LIN {X 0,Y 369.308,Z 437.482,A -85,B 0,C 180,E1 -12872.181,E2 -12872.181} C_VEL
LIN {X 0,Y 369.19,Z 437.499,A -85,B 0,C 180,E1 -12876.558,E2 -12876.558} C_VEL
LIN {X 0,Y 369.064,Z 437.51,A -85,B 0,C 180,E1 -12879.868,E2 -12879.868} C_VEL
LIN {X 0,Y 369.038,Z 437.513,A -85,B 0,C 180,E1 -12883.772,E2 -12883.772} C_VEL
LIN {X 0,Y 368.991,Z 437.518,A -85,B 0,C 180,E1 -12887.742,E2 -12887.742} C_VEL
LIN {X 0,Y 368.897,Z 437.53,A -85,B 0,C 180,E1 -12891.579,E2 -12891.579} C_VEL
LIN {X 0,Y 368.934,Z 437.529,A -85,B 0,C 180,E1 -12894.777,E2 -12894.777} C_VEL
LIN {X 0,Y 368.914,Z 437.532,A -85,B 0,C 180,E1 -12896.326,E2 -12896.326} C_VEL
LIN {X 0,Y 368.209,Z 437.626,A -85,B 0,C 180,E1 -12897.236,E2 -12897.236} C_VEL
LIN {X 0,Y 365.335,Z 437.983,A -85,B 0,C 180,E1 -12898.717,E2 -12898.717} C_VEL
LIN {X 0,Y 362.932,Z 438.276,A -85,B 0,C 180,E1 -12899.915,E2 -12899.915} C_VEL
LIN {X 0,Y 361.918,Z 438.402,A -85,B 0,C 180,E1 -12900.842,E2 -12900.842} C_VEL
LIN {X 0,Y 361.843,Z 438.409,A -85,B 0,C 180,E1 -12901.155,E2 -12901.155} C_VEL
LIN {X 0,Y 361.854,Z 438.411,A -85,B 0,C 180,E1 -12904.28,E2 -12904.28} C_VEL
LIN {X 0,Y 361.859,Z 438.407,A -85,B 0,C 180,E1 -12907.222,E2 -12907.222} C_VEL
LIN {X 0,Y 361.812,Z 438.417,A -85,B 0,C 180,E1 -12910.751,E2 -12910.751} C_VEL
LIN {X 0,Y 361.816,Z 438.416,A -85,B 0,C 180,E1 -12914.368,E2 -12914.368} C_VEL
LIN {X 0,Y 361.831,Z 438.41,A -85,B 0,C 180,E1 -12917.569,E2 -12917.569} C_VEL
LIN {X 0,Y 361.865,Z 438.408,A -85,B 0,C 180,E1 -12920.974,E2 -12920.974} C_VEL
LIN {X 0,Y 361.873,Z 438.411,A -85,B 0,C 180,E1 -12924.655,E2 -12924.655} C_VEL
LIN {X 0,Y 361.837,Z 438.413,A -85,B 0,C 180,E1 -12928.37,E2 -12928.37} C_VEL
LIN {X 0,Y 361.907,Z 438.403,A -85,B 0,C 180,E1 -12932.221,E2 -12932.221} C_VEL
LIN {X 0,Y 361.927,Z 438.404,A -85,B 0,C 180,E1 -12934.71,E2 -12934.71} C_VEL
LIN {X 0,Y 361.892,Z 438.406,A -85,B 0,C 180,E1 -12938.347,E2 -12938.347} C_VEL
LIN {X 0,Y 361.966,Z 438.394,A -85,B 0,C 180,E1 -12942.061,E2 -12942.061} C_VEL
LIN {X 0,Y 361.997,Z 438.391,A -85,B 0,C 180,E1 -12946.101,E2 -12946.101} C_VEL
LIN {X 0,Y 362.03,Z 438.386,A -85,B 0,C 180,E1 -12949.938,E2 -12949.938} C_VEL
LIN {X 0,Y 362.115,Z 438.377,A -85,B 0,C 180,E1 -12952.192,E2 -12952.192} C_VEL
LIN {X 0,Y 362.105,Z 438.38,A -85,B 0,C 180,E1 -12954.431,E2 -12954.431} C_VEL
LIN {X 0,Y 362.28,Z 438.354,A -85,B 0,C 180,E1 -12957.777,E2 -12957.777} C_VEL
LIN {X 0,Y 362.426,Z 438.337,A -85,B 0,C 180,E1 -12960,E2 -12960} C_VEL
LIN {X 0,Y 362.281,Z 438.356,A -85,B 0,C 180,E1 -12962.224,E2 -12962.224} C_VEL
LIN {X 0,Y 362.172,Z 438.374,A -85,B 0,C 180,E1 -12966.686,E2 -12966.686} C_VEL
LIN {X 0,Y 362.074,Z 438.383,A -85,B 0,C 180,E1 -12968.933,E2 -12968.933} C_VEL
LIN {X 0,Y 361.96,Z 438.397,A -85,B 0,C 180,E1 -12972.332,E2 -12972.332} C_VEL
LIN {X 0,Y 361.962,Z 438.4,A -85,B 0,C 180,E1 -12974.62,E2 -12974.62} C_VEL
LIN {X 0,Y 361.959,Z 438.395,A -85,B 0,C 180,E1 -12978.099,E2 -12978.099} C_VEL
LIN {X 0,Y 361.86,Z 438.406,A -85,B 0,C 180,E1 -12981.655,E2 -12981.655} C_VEL
LIN {X 0,Y 361.925,Z 438.399,A -85,B 0,C 180,E1 -12985.29,E2 -12985.29} C_VEL
LIN {X 0,Y 361.918,Z 438.399,A -85,B 0,C 180,E1 -12987.778,E2 -12987.778} C_VEL
LIN {X 0,Y 361.846,Z 438.409,A -85,B 0,C 180,E1 -12991.285,E2 -12991.285} C_VEL
LIN {X 0,Y 361.854,Z 438.409,A -85,B 0,C 180,E1 -12994.281,E2 -12994.281} C_VEL
LIN {X 0,Y 361.863,Z 438.408,A -85,B 0,C 180,E1 -12997.223,E2 -12997.223} C_VEL
LIN {X 0,Y 361.835,Z 438.416,A -85,B 0,C 180,E1 -13000.756,E2 -13000.756} C_VEL
LIN {X 0,Y 361.846,Z 438.411,A -85,B 0,C 180,E1 -13004.364,E2 -13004.364} C_VEL
LIN {X 0,Y 361.837,Z 438.409,A -85,B 0,C 180,E1 -13007.568,E2 -13007.568} C_VEL
LIN {X 0,Y 361.87,Z 438.409,A -85,B 0,C 180,E1 -13010.974,E2 -13010.974} C_VEL
LIN {X 0,Y 361.874,Z 438.41,A -85,B 0,C 180,E1 -13014.656,E2 -13014.656} C_VEL
LIN {X 0,Y 361.919,Z 438.421,A -85,B 0,C 180,E1 -13018.297,E2 -13018.297} C_VEL
LIN {X 0,Y 365.147,Z 453.696,A -85,B 0,C 180,E1 -13021.772,E2 -13021.772} C_VEL
LIN {X 0,Y 366.243,Z 460.205,A -85,B 0,C 180,E1 -13023.196,E2 -13023.196} C_VEL
LIN {X 0,Y 364.772,Z 476.168,A -85,B 0,C 180,E1 -13026.436,E2 -13026.436} C_VEL
LIN {X 0,Y 363.878,Z 487.411,A -85,B 0,C 180,E1 -13028.704,E2 -13028.704} C_VEL
LIN {X 0,Y 368.205,Z 525.969,A -85,B 0,C 180,E1 -13029.87,E2 -13029.87} C_VEL
LIN {X 0,Y 366.651,Z 597.039,A -85,B 0,C 180,E1 -13031.563,E2 -13031.563} C_VEL
LIN {X 0,Y 365.952,Z 610.747,A -85,B 0,C 180,E1 -13032.105,E2 -13032.105} C_VEL
LIN {X 0,Y 365.227,Z 622.771,A -85,B 0,C 180,E1 -13032.791,E2 -13032.791} C_VEL
LIN {X 0,Y 364.38,Z 633.745,A -85,B 0,C 180,E1 -13033.616,E2 -13033.616} C_VEL
LIN {X 0,Y 363.654,Z 644.048,A -85,B 0,C 180,E1 -13034.59,E2 -13034.59} C_VEL
LIN {X 0,Y 362.677,Z 655.469,A -85,B 0,C 180,E1 -13035.932,E2 -13035.932} C_VEL
LIN {X 0,Y 362.039,Z 663.558,A -85,B 0,C 180,E1 -13037.101,E2 -13037.101} C_VEL
LIN {X 0,Y 361.486,Z 671.672,A -85,B 0,C 180,E1 -13038.506,E2 -13038.506} C_VEL
LIN {X 0,Y 360.991,Z 679.552,A -85,B 0,C 180,E1 -13040.192,E2 -13040.192} C_VEL
LIN {X 0,Y 360.756,Z 684.918,A -85,B 0,C 180,E1 -13041.599,E2 -13041.599} C_VEL
LIN {X 0,Y 360.586,Z 690.069,A -85,B 0,C 180,E1 -13043.285,E2 -13043.285} C_VEL
LIN {X 0,Y 360.594,Z 694.009,A -85,B 0,C 180,E1 -13044.969,E2 -13044.969} C_VEL
LIN {X 0,Y 360.607,Z 696.828,A -85,B 0,C 180,E1 -13046.649,E2 -13046.649} C_VEL
LIN {X 0,Y 360.674,Z 698.125,A -85,B 0,C 180,E1 -13047.767,E2 -13047.767} C_VEL
LIN {X 0,Y 360.693,Z 698.989,A -85,B 0,C 180,E1 -13048.884,E2 -13048.884} C_VEL
LIN {X 0,Y 360.719,Z 699.392,A -85,B 0,C 180,E1 -13050,E2 -13050} C_VEL
LIN {X 0,Y 360.648,Z 699.335,A -85,B 0,C 180,E1 -13051.117,E2 -13051.117} C_VEL
LIN {X 0,Y 360.654,Z 698.865,A -85,B 0,C 180,E1 -13052.234,E2 -13052.234} C_VEL
LIN {X 0,Y 360.507,Z 697.964,A -85,B 0,C 180,E1 -13053.353,E2 -13053.353} C_VEL
LIN {X 0,Y 360.498,Z 696.598,A -85,B 0,C 180,E1 -13054.473,E2 -13054.473} C_VEL
LIN {X 0,Y 360.43,Z 693.966,A -85,B 0,C 180,E1 -13056.04,E2 -13056.04} C_VEL
LIN {X 0,Y 360.644,Z 689.779,A -85,B 0,C 180,E1 -13057.841,E2 -13057.841} C_VEL
LIN {X 0,Y 360.915,Z 684.658,A -85,B 0,C 180,E1 -13059.528,E2 -13059.528} C_VEL
LIN {X 0,Y 361.546,Z 677.08,A -85,B 0,C 180,E1 -13061.493,E2 -13061.493} C_VEL
LIN {X 0,Y 362.362,Z 668.888,A -85,B 0,C 180,E1 -13063.173,E2 -13063.173} C_VEL
LIN {X 0,Y 363.44,Z 659.09,A -85,B 0,C 180,E1 -13064.788,E2 -13064.788} C_VEL
LIN {X 0,Y 364.709,Z 648.239,A -85,B 0,C 180,E1 -13066.226,E2 -13066.226} C_VEL
LIN {X 0,Y 366.063,Z 636.511,A -85,B 0,C 180,E1 -13067.457,E2 -13067.457} C_VEL
LIN {X 0,Y 367.288,Z 625.218,A -85,B 0,C 180,E1 -13068.405,E2 -13068.405} C_VEL
LIN {X 0,Y 368.46,Z 612.8,A -85,B 0,C 180,E1 -13069.21,E2 -13069.21} C_VEL
LIN {X 0,Y 369.631,Z 598.545,A -85,B 0,C 180,E1 -13069.869,E2 -13069.869} C_VEL
LIN {X 0,Y 370.141,Z 584.099,A -85,B 0,C 180,E1 -13070.311,E2 -13070.311} C_VEL
LIN {X 0,Y 372.131,Z 525.028,A -85,B 0,C 180,E1 -13071.802,E2 -13071.802} C_VEL
LIN {X 0,Y 370.246,Z 506.889,A -85,B 0,C 180,E1 -13072.5,E2 -13072.5} C_VEL
LIN {X 0,Y 367.427,Z 490.28,A -85,B 0,C 180,E1 -13073.261,E2 -13073.261} C_VEL
LIN {X 0,Y 365.658,Z 481.588,A -85,B 0,C 180,E1 -13073.717,E2 -13073.717} C_VEL
LIN {X 0,Y 367.812,Z 465.224,A -85,B 0,C 180,E1 -13077.296,E2 -13077.296} C_VEL
LIN {X 0,Y 367.201,Z 460.097,A -85,B 0,C 180,E1 -13078.587,E2 -13078.587} C_VEL
LIN {X 0,Y 365.346,Z 451.385,A -85,B 0,C 180,E1 -13080.972,E2 -13080.972} C_VEL
LIN {X 0,Y 362.568,Z 440.857,A -85,B 0,C 180,E1 -13084.204,E2 -13084.204} C_VEL
LIN {X 0,Y 361.884,Z 438.415,A -85,B 0,C 180,E1 -13085.051,E2 -13085.051} C_VEL
LIN {X 0,Y 361.872,Z 438.41,A -85,B 0,C 180,E1 -13088.425,E2 -13088.425} C_VEL
LIN {X 0,Y 361.831,Z 438.416,A -85,B 0,C 180,E1 -13091.331,E2 -13091.331} C_VEL
LIN {X 0,Y 361.849,Z 438.411,A -85,B 0,C 180,E1 -13094.364,E2 -13094.364} C_VEL
LIN {X 0,Y 361.839,Z 438.411,A -85,B 0,C 180,E1 -13097.568,E2 -13097.568} C_VEL
LIN {X 0,Y 361.871,Z 438.407,A -85,B 0,C 180,E1 -13100.974,E2 -13100.974} C_VEL
LIN {X 0,Y 361.878,Z 438.408,A -85,B 0,C 180,E1 -13104.655,E2 -13104.655} C_VEL
LIN {X 0,Y 361.841,Z 438.412,A -85,B 0,C 180,E1 -13108.371,E2 -13108.371} C_VEL
LIN {X 0,Y 361.869,Z 438.408,A -85,B 0,C 180,E1 -13110.952,E2 -13110.952} C_VEL
LIN {X 0,Y 361.865,Z 438.411,A -85,B 0,C 180,E1 -13114.705,E2 -13114.705} C_VEL
LIN {X 0,Y 361.856,Z 438.412,A -85,B 0,C 180,E1 -13118.345,E2 -13118.345} C_VEL
LIN {X 0,Y 361.898,Z 438.408,A -85,B 0,C 180,E1 -13122.097,E2 -13122.097} C_VEL
LIN {X 0,Y 361.967,Z 438.399,A -85,B 0,C 180,E1 -13126.527,E2 -13126.527} C_VEL
LIN {X 0,Y 362.023,Z 438.469,A -85,B 0,C 180,E1 -13130.008,E2 -13130.008} C_VEL
LIN {X 0,Y 362.667,Z 441.065,A -85,B 0,C 180,E1 -13131.081,E2 -13131.081} C_VEL
LIN {X 0,Y 369.621,Z 454.318,A -85,B 0,C 180,E1 -13132.231,E2 -13132.231} C_VEL
LIN {X 0,Y 373.85,Z 464.17,A -85,B 0,C 180,E1 -13132.93,E2 -13132.93} C_VEL
LIN {X 0,Y 370.741,Z 546.178,A -85,B 0,C 180,E1 -13135.072,E2 -13135.072} C_VEL
LIN {X 0,Y 370.2,Z 559.452,A -85,B 0,C 180,E1 -13135.645,E2 -13135.645} C_VEL
LIN {X 0,Y 369.566,Z 570.673,A -85,B 0,C 180,E1 -13136.32,E2 -13136.32} C_VEL
LIN {X 0,Y 368.512,Z 582.778,A -85,B 0,C 180,E1 -13137.267,E2 -13137.267} C_VEL
LIN {X 0,Y 367.464,Z 593.646,A -85,B 0,C 180,E1 -13138.356,E2 -13138.356} C_VEL
LIN {X 0,Y 366.472,Z 602.547,A -85,B 0,C 180,E1 -13139.451,E2 -13139.451} C_VEL
LIN {X 0,Y 365.404,Z 611.798,A -85,B 0,C 180,E1 -13140.834,E2 -13140.834} C_VEL
LIN {X 0,Y 364.267,Z 620.676,A -85,B 0,C 180,E1 -13142.488,E2 -13142.488} C_VEL
LIN {X 0,Y 363.319,Z 627.86,A -85,B 0,C 180,E1 -13144.16,E2 -13144.16} C_VEL
LIN {X 0,Y 362.634,Z 632.731,A -85,B 0,C 180,E1 -13145.57,E2 -13145.57} C_VEL
LIN {X 0,Y 362.006,Z 637.363,A -85,B 0,C 180,E1 -13147.249,E2 -13147.249} C_VEL
LIN {X 0,Y 361.474,Z 640.889,A -85,B 0,C 180,E1 -13148.948,E2 -13148.948} C_VEL
LIN {X 0,Y 361.202,Z 642.649,A -85,B 0,C 180,E1 -13150.085,E2 -13150.085} C_VEL
LIN {X 0,Y 360.958,Z 643.938,A -85,B 0,C 180,E1 -13151.227,E2 -13151.227} C_VEL
LIN {X 0,Y 360.748,Z 645.102,A -85,B 0,C 180,E1 -13153.07,E2 -13153.07} C_VEL
LIN {X 0,Y 360.612,Z 645.184,A -85,B 0,C 180,E1 -13154.676,E2 -13154.676} C_VEL
LIN {X 0,Y 360.586,Z 644.705,A -85,B 0,C 180,E1 -13155.835,E2 -13155.835} C_VEL
LIN {X 0,Y 360.633,Z 643.471,A -85,B 0,C 180,E1 -13157.269,E2 -13157.269} C_VEL
LIN {X 0,Y 360.814,Z 640.452,A -85,B 0,C 180,E1 -13159.337,E2 -13159.337} C_VEL
LIN {X 0,Y 361.089,Z 636.357,A -85,B 0,C 180,E1 -13161.211,E2 -13161.211} C_VEL
LIN {X 0,Y 361.36,Z 631.457,A -85,B 0,C 180,E1 -13162.891,E2 -13162.891} C_VEL
LIN {X 0,Y 361.891,Z 624.786,A -85,B 0,C 180,E1 -13164.679,E2 -13164.679} C_VEL
LIN {X 0,Y 362.617,Z 616.333,A -85,B 0,C 180,E1 -13166.473,E2 -13166.473} C_VEL
LIN {X 0,Y 363.279,Z 607.449,A -85,B 0,C 180,E1 -13167.979,E2 -13167.979} C_VEL
LIN {X 0,Y 364.035,Z 597.245,A -85,B 0,C 180,E1 -13169.386,E2 -13169.386} C_VEL
LIN {X 0,Y 364.813,Z 586.918,A -85,B 0,C 180,E1 -13170.538,E2 -13170.538} C_VEL
LIN {X 0,Y 365.546,Z 575.004,A -85,B 0,C 180,E1 -13171.595,E2 -13171.595} C_VEL
LIN {X 0,Y 366.162,Z 563.718,A -85,B 0,C 180,E1 -13172.378,E2 -13172.378} C_VEL
LIN {X 0,Y 366.694,Z 550.331,A -85,B 0,C 180,E1 -13173.068,E2 -13173.068} C_VEL
LIN {X 0,Y 367.027,Z 535.975,A -85,B 0,C 180,E1 -13173.546,E2 -13173.546} C_VEL
LIN {X 0,Y 368.732,Z 457.746,A -85,B 0,C 180,E1 -13175.393,E2 -13175.393} C_VEL
LIN {X 0,Y 361.91,Z 438.405,A -85,B 0,C 180,E1 -13176.212,E2 -13176.212} C_VEL
LIN {X 0,Y 361.814,Z 438.414,A -85,B 0,C 180,E1 -13179.867,E2 -13179.867} C_VEL
LIN {X 0,Y 361.835,Z 438.412,A -85,B 0,C 180,E1 -13182.829,E2 -13182.829} C_VEL
LIN {X 0,Y 361.818,Z 438.414,A -85,B 0,C 180,E1 -13185.947,E2 -13185.947} C_VEL
LIN {X 0,Y 361.814,Z 438.412,A -85,B 0,C 180,E1 -13189.249,E2 -13189.249} C_VEL
LIN {X 0,Y 361.865,Z 438.407,A -85,B 0,C 180,E1 -13192.981,E2 -13192.981} C_VEL
LIN {X 0,Y 361.861,Z 438.411,A -85,B 0,C 180,E1 -13196.63,E2 -13196.63} C_VEL
LIN {X 0,Y 361.866,Z 438.406,A -85,B 0,C 180,E1 -13199.671,E2 -13199.671} C_VEL
LIN {X 0,Y 361.864,Z 438.406,A -85,B 0,C 180,E1 -13203.467,E2 -13203.467} C_VEL
LIN {X 0,Y 361.883,Z 438.404,A -85,B 0,C 180,E1 -13207.144,E2 -13207.144} C_VEL
LIN {X 0,Y 361.908,Z 438.404,A -85,B 0,C 180,E1 -13210.723,E2 -13210.723} C_VEL
LIN {X 0,Y 361.934,Z 438.398,A -85,B 0,C 180,E1 -13213.066,E2 -13213.066} C_VEL
LIN {X 0,Y 362.001,Z 438.395,A -85,B 0,C 180,E1 -13216.527,E2 -13216.527} C_VEL
LIN {X 0,Y 362.002,Z 438.39,A -85,B 0,C 180,E1 -13219.937,E2 -13219.937} C_VEL
LIN {X 0,Y 362.126,Z 438.373,A -85,B 0,C 180,E1 -13223.313,E2 -13223.313} C_VEL
LIN {X 0,Y 362.279,Z 438.355,A -85,B 0,C 180,E1 -13227.776,E2 -13227.776} C_VEL
LIN {X 0,Y 362.382,Z 438.343,A -85,B 0,C 180,E1 -13230,E2 -13230} C_VEL
LIN {X 0,Y 362.271,Z 438.359,A -85,B 0,C 180,E1 -13232.223,E2 -13232.223} C_VEL
LIN {X 0,Y 362.151,Z 438.375,A -85,B 0,C 180,E1 -13236.686,E2 -13236.686} C_VEL
LIN {X 0,Y 362.029,Z 438.387,A -85,B 0,C 180,E1 -13240.062,E2 -13240.062} C_VEL
LIN {X 0,Y 361.999,Z 438.39,A -85,B 0,C 180,E1 -13243.898,E2 -13243.898} C_VEL
LIN {X 0,Y 361.929,Z 438.4,A -85,B 0,C 180,E1 -13246.934,E2 -13246.934} C_VEL
LIN {X 0,Y 361.887,Z 438.409,A -85,B 0,C 180,E1 -13250.461,E2 -13250.461} C_VEL
LIN {X 0,Y 361.893,Z 438.405,A -85,B 0,C 180,E1 -13254.112,E2 -13254.112} C_VEL
LIN {X 0,Y 361.849,Z 438.408,A -85,B 0,C 180,E1 -13257.784,E2 -13257.784} C_VEL
LIN {X 0,Y 361.843,Z 438.409,A -85,B 0,C 180,E1 -13261.155,E2 -13261.155} C_VEL
LIN {X 0,Y 361.198,Z 438.493,A -85,B 0,C 180,E1 -13262.084,E2 -13262.084} C_VEL
LIN {X 0,Y 358.363,Z 438.842,A -85,B 0,C 180,E1 -13263.593,E2 -13263.593} C_VEL
LIN {X 0,Y 355.942,Z 439.147,A -85,B 0,C 180,E1 -13264.814,E2 -13264.814} C_VEL
LIN {X 0,Y 354.891,Z 439.275,A -85,B 0,C 180,E1 -13265.759,E2 -13265.759} C_VEL
LIN {X 0,Y 354.801,Z 439.288,A -85,B 0,C 180,E1 -13266.079,E2 -13266.079} C_VEL
LIN {X 0,Y 354.767,Z 439.29,A -85,B 0,C 180,E1 -13269.412,E2 -13269.412} C_VEL
LIN {X 0,Y 354.784,Z 439.291,A -85,B 0,C 180,E1 -13272.866,E2 -13272.866} C_VEL
LIN {X 0,Y 354.766,Z 439.292,A -85,B 0,C 180,E1 -13276.103,E2 -13276.103} C_VEL
LIN {X 0,Y 354.781,Z 439.289,A -85,B 0,C 180,E1 -13279.178,E2 -13279.178} C_VEL
LIN {X 0,Y 354.805,Z 439.29,A -85,B 0,C 180,E1 -13282.403,E2 -13282.403} C_VEL
LIN {X 0,Y 354.811,Z 439.287,A -85,B 0,C 180,E1 -13284.941,E2 -13284.941} C_VEL
LIN {X 0,Y 354.792,Z 439.291,A -85,B 0,C 180,E1 -13288.405,E2 -13288.405} C_VEL
LIN {X 0,Y 354.845,Z 439.28,A -85,B 0,C 180,E1 -13291.619,E2 -13291.619} C_VEL
LIN {X 0,Y 354.898,Z 439.276,A -85,B 0,C 180,E1 -13294.172,E2 -13294.172} C_VEL
LIN {X 0,Y 354.835,Z 439.282,A -85,B 0,C 180,E1 -13297.894,E2 -13297.894} C_VEL
LIN {X 0,Y 354.921,Z 439.271,A -85,B 0,C 180,E1 -13301.892,E2 -13301.892} C_VEL
LIN {X 0,Y 354.942,Z 439.269,A -85,B 0,C 180,E1 -13305.981,E2 -13305.981} C_VEL
LIN {X 0,Y 354.977,Z 439.264,A -85,B 0,C 180,E1 -13309.736,E2 -13309.736} C_VEL
LIN {X 0,Y 355.079,Z 439.252,A -85,B 0,C 180,E1 -13312.036,E2 -13312.036} C_VEL
LIN {X 0,Y 355.079,Z 439.254,A -85,B 0,C 180,E1 -13314.321,E2 -13314.321} C_VEL
LIN {X 0,Y 355.243,Z 439.231,A -85,B 0,C 180,E1 -13317.732,E2 -13317.732} C_VEL
LIN {X 0,Y 355.395,Z 439.212,A -85,B 0,C 180,E1 -13320,E2 -13320} C_VEL
LIN {X 0,Y 355.244,Z 439.233,A -85,B 0,C 180,E1 -13322.268,E2 -13322.268} C_VEL
LIN {X 0,Y 355.138,Z 439.249,A -85,B 0,C 180,E1 -13326.819,E2 -13326.819} C_VEL
LIN {X 0,Y 355.015,Z 439.261,A -85,B 0,C 180,E1 -13329.112,E2 -13329.112} C_VEL
LIN {X 0,Y 354.921,Z 439.276,A -85,B 0,C 180,E1 -13332.581,E2 -13332.581} C_VEL
LIN {X 0,Y 354.889,Z 439.276,A -85,B 0,C 180,E1 -13336.096,E2 -13336.096} C_VEL
LIN {X 0,Y 354.906,Z 439.277,A -85,B 0,C 180,E1 -13338.472,E2 -13338.472} C_VEL
LIN {X 0,Y 354.815,Z 439.285,A -85,B 0,C 180,E1 -13342.107,E2 -13342.107} C_VEL
LIN {X 0,Y 354.897,Z 439.274,A -85,B 0,C 180,E1 -13345.828,E2 -13345.828} C_VEL
LIN {X 0,Y 354.853,Z 439.279,A -85,B 0,C 180,E1 -13349.679,E2 -13349.679} C_VEL
LIN {X 0,Y 354.806,Z 439.285,A -85,B 0,C 180,E1 -13353.702,E2 -13353.702} C_VEL
LIN {X 0,Y 354.798,Z 439.29,A -85,B 0,C 180,E1 -13356.46,E2 -13356.46} C_VEL
LIN {X 0,Y 354.824,Z 439.284,A -85,B 0,C 180,E1 -13359.424,E2 -13359.424} C_VEL
LIN {X 0,Y 354.788,Z 439.292,A -85,B 0,C 180,E1 -13362.868,E2 -13362.868} C_VEL
LIN {X 0,Y 354.769,Z 439.291,A -85,B 0,C 180,E1 -13366.104,E2 -13366.104} C_VEL
LIN {X 0,Y 354.789,Z 439.289,A -85,B 0,C 180,E1 -13369.18,E2 -13369.18} C_VEL
LIN {X 0,Y 354.807,Z 439.288,A -85,B 0,C 180,E1 -13372.403,E2 -13372.403} C_VEL
LIN {X 0,Y 354.812,Z 439.29,A -85,B 0,C 180,E1 -13374.941,E2 -13374.941} C_VEL
LIN {X 0,Y 354.89,Z 439.481,A -85,B 0,C 180,E1 -13378.073,E2 -13378.073} C_VEL
LIN {X 0,Y 358.428,Z 456.128,A -85,B 0,C 180,E1 -13381.928,E2 -13381.928} C_VEL
LIN {X 0,Y 359.247,Z 460.678,A -85,B 0,C 180,E1 -13382.946,E2 -13382.946} C_VEL
LIN {X 0,Y 358.232,Z 472.293,A -85,B 0,C 180,E1 -13385.362,E2 -13385.362} C_VEL
LIN {X 0,Y 356.947,Z 487.261,A -85,B 0,C 180,E1 -13388.393,E2 -13388.393} C_VEL
LIN {X 0,Y 361.36,Z 526.178,A -85,B 0,C 180,E1 -13389.59,E2 -13389.59} C_VEL
LIN {X 0,Y 359.711,Z 597.137,A -85,B 0,C 180,E1 -13391.342,E2 -13391.342} C_VEL
LIN {X 0,Y 358.975,Z 610.596,A -85,B 0,C 180,E1 -13391.893,E2 -13391.893} C_VEL
LIN {X 0,Y 358.257,Z 622.505,A -85,B 0,C 180,E1 -13392.593,E2 -13392.593} C_VEL
LIN {X 0,Y 357.392,Z 633.414,A -85,B 0,C 180,E1 -13393.433,E2 -13393.433} C_VEL
LIN {X 0,Y 356.603,Z 643.672,A -85,B 0,C 180,E1 -13394.424,E2 -13394.424} C_VEL
LIN {X 0,Y 355.689,Z 654.044,A -85,B 0,C 180,E1 -13395.658,E2 -13395.658} C_VEL
LIN {X 0,Y 355.086,Z 662.242,A -85,B 0,C 180,E1 -13396.844,E2 -13396.844} C_VEL
LIN {X 0,Y 354.492,Z 670.487,A -85,B 0,C 180,E1 -13398.276,E2 -13398.276} C_VEL
LIN {X 0,Y 353.932,Z 678.527,A -85,B 0,C 180,E1 -13399.995,E2 -13399.995} C_VEL
LIN {X 0,Y 353.681,Z 683.982,A -85,B 0,C 180,E1 -13401.43,E2 -13401.43} C_VEL
LIN {X 0,Y 353.51,Z 689.226,A -85,B 0,C 180,E1 -13403.15,E2 -13403.15} C_VEL
LIN {X 0,Y 353.527,Z 693.245,A -85,B 0,C 180,E1 -13404.868,E2 -13404.868} C_VEL
LIN {X 0,Y 353.52,Z 696.132,A -85,B 0,C 180,E1 -13406.581,E2 -13406.581} C_VEL
LIN {X 0,Y 353.609,Z 697.464,A -85,B 0,C 180,E1 -13407.722,E2 -13407.722} C_VEL
LIN {X 0,Y 353.621,Z 698.357,A -85,B 0,C 180,E1 -13408.862,E2 -13408.862} C_VEL
LIN {X 0,Y 353.643,Z 698.814,A -85,B 0,C 180,E1 -13410,E2 -13410} C_VEL
LIN {X 0,Y 353.579,Z 698.788,A -85,B 0,C 180,E1 -13411.139,E2 -13411.139} C_VEL
LIN {X 0,Y 353.585,Z 698.341,A -85,B 0,C 180,E1 -13412.279,E2 -13412.279} C_VEL
LIN {X 0,Y 353.416,Z 697.464,A -85,B 0,C 180,E1 -13413.421,E2 -13413.421} C_VEL
LIN {X 0,Y 353.423,Z 696.145,A -85,B 0,C 180,E1 -13414.563,E2 -13414.563} C_VEL
LIN {X 0,Y 353.336,Z 693.839,A -85,B 0,C 180,E1 -13415.998,E2 -13415.998} C_VEL
LIN {X 0,Y 353.559,Z 689.44,A -85,B 0,C 180,E1 -13417.999,E2 -13417.999} C_VEL
LIN {X 0,Y 353.894,Z 684.404,A -85,B 0,C 180,E1 -13419.719,E2 -13419.719} C_VEL
LIN {X 0,Y 354.409,Z 678.075,A -85,B 0,C 180,E1 -13421.438,E2 -13421.438} C_VEL
LIN {X 0,Y 355.277,Z 670.24,A -85,B 0,C 180,E1 -13423.15,E2 -13423.15} C_VEL
LIN {X 0,Y 356.412,Z 660.562,A -85,B 0,C 180,E1 -13424.854,E2 -13424.854} C_VEL
LIN {X 0,Y 357.746,Z 649.562,A -85,B 0,C 180,E1 -13426.404,E2 -13426.404} C_VEL
LIN {X 0,Y 359.115,Z 638.449,A -85,B 0,C 180,E1 -13427.659,E2 -13427.659} C_VEL
LIN {X 0,Y 360.588,Z 625.985,A -85,B 0,C 180,E1 -13428.76,E2 -13428.76} C_VEL
LIN {X 0,Y 361.807,Z 614.063,A -85,B 0,C 180,E1 -13429.578,E2 -13429.578} C_VEL
LIN {X 0,Y 363.006,Z 600.605,A -85,B 0,C 180,E1 -13430.248,E2 -13430.248} C_VEL
LIN {X 0,Y 363.672,Z 586.618,A -85,B 0,C 180,E1 -13430.726,E2 -13430.726} C_VEL
LIN {X 0,Y 365.896,Z 526.081,A -85,B 0,C 180,E1 -13432.306,E2 -13432.306} C_VEL
LIN {X 0,Y 364.139,Z 508.606,A -85,B 0,C 180,E1 -13432.999,E2 -13432.999} C_VEL
LIN {X 0,Y 361.28,Z 491.374,A -85,B 0,C 180,E1 -13433.817,E2 -13433.817} C_VEL
LIN {X 0,Y 359.148,Z 480.74,A -85,B 0,C 180,E1 -13434.418,E2 -13434.418} C_VEL
LIN {X 0,Y 361.078,Z 466.886,A -85,B 0,C 180,E1 -13437.534,E2 -13437.534} C_VEL
LIN {X 0,Y 360.187,Z 460.544,A -85,B 0,C 180,E1 -13439.197,E2 -13439.197} C_VEL
LIN {X 0,Y 358.274,Z 452.029,A -85,B 0,C 180,E1 -13441.651,E2 -13441.651} C_VEL
LIN {X 0,Y 356.049,Z 443.564,A -85,B 0,C 180,E1 -13444.356,E2 -13444.356} C_VEL
LIN {X 0,Y 354.827,Z 439.291,A -85,B 0,C 180,E1 -13445.869,E2 -13445.869} C_VEL
LIN {X 0,Y 354.827,Z 439.286,A -85,B 0,C 180,E1 -13449.424,E2 -13449.424} C_VEL
LIN {X 0,Y 354.792,Z 439.293,A -85,B 0,C 180,E1 -13452.868,E2 -13452.868} C_VEL
LIN {X 0,Y 354.771,Z 439.292,A -85,B 0,C 180,E1 -13456.104,E2 -13456.104} C_VEL
LIN {X 0,Y 354.79,Z 439.289,A -85,B 0,C 180,E1 -13459.179,E2 -13459.179} C_VEL
LIN {X 0,Y 354.814,Z 439.29,A -85,B 0,C 180,E1 -13462.402,E2 -13462.402} C_VEL
LIN {X 0,Y 354.815,Z 439.285,A -85,B 0,C 180,E1 -13464.941,E2 -13464.941} C_VEL
LIN {X 0,Y 354.797,Z 439.29,A -85,B 0,C 180,E1 -13468.405,E2 -13468.405} C_VEL
LIN {X 0,Y 354.802,Z 439.287,A -85,B 0,C 180,E1 -13471.615,E2 -13471.615} C_VEL
LIN {X 0,Y 354.807,Z 439.288,A -85,B 0,C 180,E1 -13475.42,E2 -13475.42} C_VEL
LIN {X 0,Y 354.821,Z 439.287,A -85,B 0,C 180,E1 -13479.113,E2 -13479.113} C_VEL
LIN {X 0,Y 354.84,Z 439.284,A -85,B 0,C 180,E1 -13482.717,E2 -13482.717} C_VEL
LIN {X 0,Y 354.911,Z 439.278,A -85,B 0,C 180,E1 -13486.253,E2 -13486.253} C_VEL
LIN {X 0,Y 354.914,Z 439.292,A -85,B 0,C 180,E1 -13489.157,E2 -13489.157} C_VEL
LIN {X 0,Y 355.636,Z 442.015,A -85,B 0,C 180,E1 -13490.331,E2 -13490.331} C_VEL
LIN {X 0,Y 362.996,Z 455.484,A -85,B 0,C 180,E1 -13491.597,E2 -13491.597} C_VEL
LIN {X 0,Y 367.479,Z 465.649,A -85,B 0,C 180,E1 -13492.382,E2 -13492.382} C_VEL
LIN {X 0,Y 367.577,Z 468.483,A -85,B 0,C 180,E1 -13492.478,E2 -13492.478} C_VEL
LIN {X 0,Y 364.432,Z 546.454,A -85,B 0,C 180,E1 -13494.571,E2 -13494.571} C_VEL
LIN {X 0,Y 363.821,Z 559.719,A -85,B 0,C 180,E1 -13495.152,E2 -13495.152} C_VEL
LIN {X 0,Y 363.02,Z 572.859,A -85,B 0,C 180,E1 -13495.976,E2 -13495.976} C_VEL
LIN {X 0,Y 361.911,Z 584.649,A -85,B 0,C 180,E1 -13496.939,E2 -13496.939} C_VEL
LIN {X 0,Y 360.819,Z 595.309,A -85,B 0,C 180,E1 -13498.047,E2 -13498.047} C_VEL
LIN {X 0,Y 359.505,Z 605.986,A -85,B 0,C 180,E1 -13499.44,E2 -13499.44} C_VEL
LIN {X 0,Y 358.47,Z 614.632,A -85,B 0,C 180,E1 -13500.844,E2 -13500.844} C_VEL
LIN {X 0,Y 357.436,Z 621.819,A -85,B 0,C 180,E1 -13502.254,E2 -13502.254} C_VEL
LIN {X 0,Y 356.418,Z 628.887,A -85,B 0,C 180,E1 -13503.957,E2 -13503.957} C_VEL
LIN {X 0,Y 355.58,Z 634.509,A -85,B 0,C 180,E1 -13505.671,E2 -13505.671} C_VEL
LIN {X 0,Y 354.956,Z 638.79,A -85,B 0,C 180,E1 -13507.35,E2 -13507.35} C_VEL
LIN {X 0,Y 354.383,Z 642.155,A -85,B 0,C 180,E1 -13509.129,E2 -13509.129} C_VEL
LIN {X 0,Y 354.107,Z 643.741,A -85,B 0,C 180,E1 -13510.29,E2 -13510.29} C_VEL
LIN {X 0,Y 353.86,Z 644.906,A -85,B 0,C 180,E1 -13511.456,E2 -13511.456} C_VEL
LIN {X 0,Y 353.675,Z 645.764,A -85,B 0,C 180,E1 -13513.168,E2 -13513.168} C_VEL
LIN {X 0,Y 353.517,Z 645.654,A -85,B 0,C 180,E1 -13514.978,E2 -13514.978} C_VEL
LIN {X 0,Y 353.535,Z 644.999,A -85,B 0,C 180,E1 -13516.159,E2 -13516.159} C_VEL
LIN {X 0,Y 353.566,Z 643.795,A -85,B 0,C 180,E1 -13517.421,E2 -13517.421} C_VEL
LIN {X 0,Y 353.707,Z 641.312,A -85,B 0,C 180,E1 -13519.138,E2 -13519.138} C_VEL
LIN {X 0,Y 353.966,Z 637.306,A -85,B 0,C 180,E1 -13521.062,E2 -13521.062} C_VEL
LIN {X 0,Y 354.343,Z 631.576,A -85,B 0,C 180,E1 -13523.062,E2 -13523.062} C_VEL
LIN {X 0,Y 354.892,Z 624.782,A -85,B 0,C 180,E1 -13524.886,E2 -13524.886} C_VEL
LIN {X 0,Y 355.511,Z 617.737,A -85,B 0,C 180,E1 -13526.41,E2 -13526.41} C_VEL
LIN {X 0,Y 356.182,Z 608.85,A -85,B 0,C 180,E1 -13527.981,E2 -13527.981} C_VEL
LIN {X 0,Y 356.996,Z 598.287,A -85,B 0,C 180,E1 -13529.483,E2 -13529.483} C_VEL
LIN {X 0,Y 357.825,Z 587.586,A -85,B 0,C 180,E1 -13530.708,E2 -13530.708} C_VEL
LIN {X 0,Y 358.586,Z 575.709,A -85,B 0,C 180,E1 -13531.785,E2 -13531.785} C_VEL
LIN {X 0,Y 359.274,Z 563.374,A -85,B 0,C 180,E1 -13532.653,E2 -13532.653} C_VEL
LIN {X 0,Y 359.781,Z 550.273,A -85,B 0,C 180,E1 -13533.326,E2 -13533.326} C_VEL
LIN {X 0,Y 360.117,Z 536.424,A -85,B 0,C 180,E1 -13533.794,E2 -13533.794} C_VEL
LIN {X 0,Y 361.9,Z 459.291,A -85,B 0,C 180,E1 -13535.658,E2 -13535.658} C_VEL
LIN {X 0,Y 354.853,Z 439.284,A -85,B 0,C 180,E1 -13536.519,E2 -13536.519} C_VEL
LIN {X 0,Y 354.77,Z 439.29,A -85,B 0,C 180,E1 -13539.412,E2 -13539.412} C_VEL
LIN {X 0,Y 354.787,Z 439.289,A -85,B 0,C 180,E1 -13542.866,E2 -13542.866} C_VEL
LIN {X 0,Y 354.767,Z 439.293,A -85,B 0,C 180,E1 -13546.103,E2 -13546.103} C_VEL
LIN {X 0,Y 354.767,Z 439.29,A -85,B 0,C 180,E1 -13549.175,E2 -13549.175} C_VEL
LIN {X 0,Y 354.801,Z 439.292,A -85,B 0,C 180,E1 -13552.404,E2 -13552.404} C_VEL
LIN {X 0,Y 354.813,Z 439.286,A -85,B 0,C 180,E1 -13554.94,E2 -13554.94} C_VEL
LIN {X 0,Y 354.796,Z 439.293,A -85,B 0,C 180,E1 -13558.405,E2 -13558.405} C_VEL
LIN {X 0,Y 354.801,Z 439.286,A -85,B 0,C 180,E1 -13561.614,E2 -13561.614} C_VEL
LIN {X 0,Y 354.836,Z 439.282,A -85,B 0,C 180,E1 -13565.657,E2 -13565.657} C_VEL
LIN {X 0,Y 354.842,Z 439.281,A -85,B 0,C 180,E1 -13569.114,E2 -13569.114} C_VEL
LIN {X 0,Y 354.9,Z 439.277,A -85,B 0,C 180,E1 -13572.72,E2 -13572.72} C_VEL
LIN {X 0,Y 354.953,Z 439.271,A -85,B 0,C 180,E1 -13576.255,E2 -13576.255} C_VEL
LIN {X 0,Y 354.958,Z 439.267,A -85,B 0,C 180,E1 -13579.735,E2 -13579.735} C_VEL
LIN {X 0,Y 355.091,Z 439.25,A -85,B 0,C 180,E1 -13583.179,E2 -13583.179} C_VEL
LIN {X 0,Y 355.242,Z 439.231,A -85,B 0,C 180,E1 -13587.732,E2 -13587.732} C_VEL
LIN {X 0,Y 355.333,Z 439.221,A -85,B 0,C 180,E1 -13590,E2 -13590} C_VEL
LIN {X 0,Y 355.234,Z 439.236,A -85,B 0,C 180,E1 -13592.267,E2 -13592.267} C_VEL
LIN {X 0,Y 355.114,Z 439.25,A -85,B 0,C 180,E1 -13596.819,E2 -13596.819} C_VEL
LIN {X 0,Y 354.976,Z 439.268,A -85,B 0,C 180,E1 -13600.264,E2 -13600.264} C_VEL
LIN {X 0,Y 354.944,Z 439.27,A -85,B 0,C 180,E1 -13604.019,E2 -13604.019} C_VEL
LIN {X 0,Y 354.89,Z 439.277,A -85,B 0,C 180,E1 -13608.092,E2 -13608.092} C_VEL
LIN {X 0,Y 354.815,Z 439.286,A -85,B 0,C 180,E1 -13612.107,E2 -13612.107} C_VEL
LIN {X 0,Y 354.851,Z 439.286,A -85,B 0,C 180,E1 -13614.577,E2 -13614.577} C_VEL
LIN {X 0,Y 354.802,Z 439.29,A -85,B 0,C 180,E1 -13618.385,E2 -13618.385} C_VEL
LIN {X 0,Y 354.786,Z 439.292,A -85,B 0,C 180,E1 -13622.333,E2 -13622.333} C_VEL
LIN {X 0,Y 354.801,Z 439.288,A -85,B 0,C 180,E1 -13626.079,E2 -13626.079} C_VEL
LIN {X 0,Y 354.106,Z 439.379,A -85,B 0,C 180,E1 -13627.026,E2 -13627.026} C_VEL
LIN {X 0,Y 351.207,Z 439.74,A -85,B 0,C 180,E1 -13628.566,E2 -13628.566} C_VEL
LIN {X 0,Y 348.781,Z 440.038,A -85,B 0,C 180,E1 -13629.812,E2 -13629.812} C_VEL
LIN {X 0,Y 347.77,Z 440.166,A -85,B 0,C 180,E1 -13630.777,E2 -13630.777} C_VEL
LIN {X 0,Y 347.703,Z 440.169,A -85,B 0,C 180,E1 -13631.104,E2 -13631.104} C_VEL
LIN {X 0,Y 347.721,Z 440.168,A -85,B 0,C 180,E1 -13633.408,E2 -13633.408} C_VEL
LIN {X 0,Y 347.724,Z 440.173,A -85,B 0,C 180,E1 -13636.686,E2 -13636.686} C_VEL
LIN {X 0,Y 347.744,Z 440.167,A -85,B 0,C 180,E1 -13640.173,E2 -13640.173} C_VEL
LIN {X 0,Y 347.76,Z 440.168,A -85,B 0,C 180,E1 -13642.679,E2 -13642.679} C_VEL
LIN {X 0,Y 347.747,Z 440.165,A -85,B 0,C 180,E1 -13645.956,E2 -13645.956} C_VEL
LIN {X 0,Y 347.748,Z 440.164,A -85,B 0,C 180,E1 -13649.652,E2 -13649.652} C_VEL
LIN {X 0,Y 347.829,Z 440.154,A -85,B 0,C 180,E1 -13653.608,E2 -13653.608} C_VEL
LIN {X 0,Y 347.788,Z 440.161,A -85,B 0,C 180,E1 -13656.162,E2 -13656.162} C_VEL
LIN {X 0,Y 347.812,Z 440.157,A -85,B 0,C 180,E1 -13659.909,E2 -13659.909} C_VEL
LIN {X 0,Y 347.865,Z 440.153,A -85,B 0,C 180,E1 -13662.359,E2 -13662.359} C_VEL
LIN {X 0,Y 347.896,Z 440.147,A -85,B 0,C 180,E1 -13665.971,E2 -13665.971} C_VEL
LIN {X 0,Y 347.928,Z 440.142,A -85,B 0,C 180,E1 -13669.526,E2 -13669.526} C_VEL
LIN {X 0,Y 348.043,Z 440.128,A -85,B 0,C 180,E1 -13671.874,E2 -13671.874} C_VEL
LIN {X 0,Y 348.054,Z 440.128,A -85,B 0,C 180,E1 -13674.206,E2 -13674.206} C_VEL
LIN {X 0,Y 348.205,Z 440.107,A -85,B 0,C 180,E1 -13677.687,E2 -13677.687} C_VEL
LIN {X 0,Y 348.344,Z 440.091,A -85,B 0,C 180,E1 -13680,E2 -13680} C_VEL
LIN {X 0,Y 348.206,Z 440.11,A -85,B 0,C 180,E1 -13682.314,E2 -13682.314} C_VEL
LIN {X 0,Y 348.106,Z 440.123,A -85,B 0,C 180,E1 -13686.958,E2 -13686.958} C_VEL
LIN {X 0,Y 347.967,Z 440.138,A -85,B 0,C 180,E1 -13689.299,E2 -13689.299} C_VEL
LIN {X 0,Y 347.889,Z 440.151,A -85,B 0,C 180,E1 -13692.84,E2 -13692.84} C_VEL
LIN {X 0,Y 347.839,Z 440.157,A -85,B 0,C 180,E1 -13696.431,E2 -13696.431} C_VEL
LIN {X 0,Y 347.855,Z 440.156,A -85,B 0,C 180,E1 -13698.86,E2 -13698.86} C_VEL
LIN {X 0,Y 347.761,Z 440.168,A -85,B 0,C 180,E1 -13702.58,E2 -13702.58} C_VEL
LIN {X 0,Y 347.81,Z 440.159,A -85,B 0,C 180,E1 -13705.109,E2 -13705.109} C_VEL
LIN {X 0,Y 347.81,Z 440.157,A -85,B 0,C 180,E1 -13707.694,E2 -13707.694} C_VEL
LIN {X 0,Y 347.763,Z 440.165,A -85,B 0,C 180,E1 -13710.347,E2 -13710.347} C_VEL
LIN {X 0,Y 347.744,Z 440.169,A -85,B 0,C 180,E1 -13714.464,E2 -13714.464} C_VEL
LIN {X 0,Y 347.773,Z 440.162,A -85,B 0,C 180,E1 -13717.989,E2 -13717.989} C_VEL
LIN {X 0,Y 347.75,Z 440.164,A -85,B 0,C 180,E1 -13721.831,E2 -13721.831} C_VEL
LIN {X 0,Y 347.766,Z 440.166,A -85,B 0,C 180,E1 -13725.017,E2 -13725.017} C_VEL
LIN {X 0,Y 347.751,Z 440.167,A -85,B 0,C 180,E1 -13728.397,E2 -13728.397} C_VEL
LIN {X 0,Y 347.774,Z 440.162,A -85,B 0,C 180,E1 -13732.012,E2 -13732.012} C_VEL
LIN {X 0,Y 347.745,Z 440.167,A -85,B 0,C 180,E1 -13735.537,E2 -13735.537} C_VEL
LIN {X 0,Y 347.802,Z 440.275,A -85,B 0,C 180,E1 -13737.781,E2 -13737.781} C_VEL
LIN {X 0,Y 351.319,Z 456.69,A -85,B 0,C 180,E1 -13741.667,E2 -13741.667} C_VEL
LIN {X 0,Y 352.254,Z 462.597,A -85,B 0,C 180,E1 -13743.006,E2 -13743.006} C_VEL
LIN {X 0,Y 350.422,Z 481.514,A -85,B 0,C 180,E1 -13746.996,E2 -13746.996} C_VEL
LIN {X 0,Y 349.985,Z 486.472,A -85,B 0,C 180,E1 -13748.037,E2 -13748.037} C_VEL
LIN {X 0,Y 354.467,Z 527.02,A -85,B 0,C 180,E1 -13749.33,E2 -13749.33} C_VEL
LIN {X 0,Y 352.765,Z 596.13,A -85,B 0,C 180,E1 -13751.073,E2 -13751.073} C_VEL
LIN {X 0,Y 352.037,Z 609.711,A -85,B 0,C 180,E1 -13751.636,E2 -13751.636} C_VEL
LIN {X 0,Y 351.291,Z 622.231,A -85,B 0,C 180,E1 -13752.387,E2 -13752.387} C_VEL
LIN {X 0,Y 350.407,Z 633.083,A -85,B 0,C 180,E1 -13753.243,E2 -13753.243} C_VEL
LIN {X 0,Y 349.535,Z 644.622,A -85,B 0,C 180,E1 -13754.4,E2 -13754.4} C_VEL
LIN {X 0,Y 348.523,Z 655.487,A -85,B 0,C 180,E1 -13755.761,E2 -13755.761} C_VEL
LIN {X 0,Y 347.94,Z 662.742,A -85,B 0,C 180,E1 -13756.866,E2 -13756.866} C_VEL
LIN {X 0,Y 347.366,Z 670.821,A -85,B 0,C 180,E1 -13758.328,E2 -13758.328} C_VEL
LIN {X 0,Y 346.834,Z 678.659,A -85,B 0,C 180,E1 -13760.082,E2 -13760.082} C_VEL
LIN {X 0,Y 346.556,Z 684.933,A -85,B 0,C 180,E1 -13761.839,E2 -13761.839} C_VEL
LIN {X 0,Y 346.426,Z 690.27,A -85,B 0,C 180,E1 -13763.759,E2 -13763.759} C_VEL
LIN {X 0,Y 346.419,Z 693.564,A -85,B 0,C 180,E1 -13765.346,E2 -13765.346} C_VEL
LIN {X 0,Y 346.434,Z 695.434,A -85,B 0,C 180,E1 -13766.511,E2 -13766.511} C_VEL
LIN {X 0,Y 346.545,Z 696.802,A -85,B 0,C 180,E1 -13767.676,E2 -13767.676} C_VEL
LIN {X 0,Y 346.552,Z 697.724,A -85,B 0,C 180,E1 -13768.838,E2 -13768.838} C_VEL
LIN {X 0,Y 346.57,Z 698.222,A -85,B 0,C 180,E1 -13770,E2 -13770} C_VEL
LIN {X 0,Y 346.512,Z 698.24,A -85,B 0,C 180,E1 -13771.163,E2 -13771.163} C_VEL
LIN {X 0,Y 346.498,Z 697.818,A -85,B 0,C 180,E1 -13772.325,E2 -13772.325} C_VEL
LIN {X 0,Y 346.329,Z 696.969,A -85,B 0,C 180,E1 -13773.491,E2 -13773.491} C_VEL
LIN {X 0,Y 346.325,Z 695.704,A -85,B 0,C 180,E1 -13774.656,E2 -13774.656} C_VEL
LIN {X 0,Y 346.243,Z 693.724,A -85,B 0,C 180,E1 -13775.957,E2 -13775.957} C_VEL
LIN {X 0,Y 346.5,Z 689.111,A -85,B 0,C 180,E1 -13778.163,E2 -13778.163} C_VEL
LIN {X 0,Y 346.856,Z 684.143,A -85,B 0,C 180,E1 -13779.918,E2 -13779.918} C_VEL
LIN {X 0,Y 347.424,Z 677.88,A -85,B 0,C 180,E1 -13781.671,E2 -13781.671} C_VEL
LIN {X 0,Y 348.34,Z 670.162,A -85,B 0,C 180,E1 -13783.417,E2 -13783.417} C_VEL
LIN {X 0,Y 349.546,Z 660.499,A -85,B 0,C 180,E1 -13785.183,E2 -13785.183} C_VEL
LIN {X 0,Y 350.964,Z 649.827,A -85,B 0,C 180,E1 -13786.73,E2 -13786.73} C_VEL
LIN {X 0,Y 352.383,Z 638.901,A -85,B 0,C 180,E1 -13788.008,E2 -13788.008} C_VEL
LIN {X 0,Y 353.91,Z 626.75,A -85,B 0,C 180,E1 -13789.127,E2 -13789.127} C_VEL
LIN {X 0,Y 355.301,Z 614.179,A -85,B 0,C 180,E1 -13790.027,E2 -13790.027} C_VEL
LIN {X 0,Y 356.555,Z 601.303,A -85,B 0,C 180,E1 -13790.706,E2 -13790.706} C_VEL
LIN {X 0,Y 357.325,Z 587.057,A -85,B 0,C 180,E1 -13791.225,E2 -13791.225} C_VEL
LIN {X 0,Y 359.683,Z 526.836,A -85,B 0,C 180,E1 -13792.841,E2 -13792.841} C_VEL
LIN {X 0,Y 358.079,Z 510.117,A -85,B 0,C 180,E1 -13793.53,E2 -13793.53} C_VEL
LIN {X 0,Y 355.414,Z 493.553,A -85,B 0,C 180,E1 -13794.351,E2 -13794.351} C_VEL
LIN {X 0,Y 352.643,Z 480.019,A -85,B 0,C 180,E1 -13795.135,E2 -13795.135} C_VEL
LIN {X 0,Y 354.36,Z 468.584,A -85,B 0,C 180,E1 -13797.78,E2 -13797.78} C_VEL
LIN {X 0,Y 353.215,Z 461.109,A -85,B 0,C 180,E1 -13799.831,E2 -13799.831} C_VEL
LIN {X 0,Y 350.958,Z 451.546,A -85,B 0,C 180,E1 -13802.748,E2 -13802.748} C_VEL
LIN {X 0,Y 348.838,Z 443.855,A -85,B 0,C 180,E1 -13805.396,E2 -13805.396} C_VEL
LIN {X 0,Y 347.77,Z 440.168,A -85,B 0,C 180,E1 -13806.811,E2 -13806.811} C_VEL
LIN {X 0,Y 347.736,Z 440.171,A -85,B 0,C 180,E1 -13810.297,E2 -13810.297} C_VEL
LIN {X 0,Y 347.73,Z 440.17,A -85,B 0,C 180,E1 -13813.408,E2 -13813.408} C_VEL
LIN {X 0,Y 347.729,Z 440.172,A -85,B 0,C 180,E1 -13816.686,E2 -13816.686} C_VEL
LIN {X 0,Y 347.75,Z 440.168,A -85,B 0,C 180,E1 -13820.173,E2 -13820.173} C_VEL
LIN {X 0,Y 347.768,Z 440.166,A -85,B 0,C 180,E1 -13822.68,E2 -13822.68} C_VEL
LIN {X 0,Y 347.752,Z 440.164,A -85,B 0,C 180,E1 -13825.956,E2 -13825.956} C_VEL
LIN {X 0,Y 347.744,Z 440.165,A -85,B 0,C 180,E1 -13829.651,E2 -13829.651} C_VEL
LIN {X 0,Y 347.746,Z 440.166,A -85,B 0,C 180,E1 -13833.601,E2 -13833.601} C_VEL
LIN {X 0,Y 347.752,Z 440.167,A -85,B 0,C 180,E1 -13836.159,E2 -13836.159} C_VEL
LIN {X 0,Y 347.743,Z 440.168,A -85,B 0,C 180,E1 -13839.905,E2 -13839.905} C_VEL
LIN {X 0,Y 347.8,Z 440.162,A -85,B 0,C 180,E1 -13842.356,E2 -13842.356} C_VEL
LIN {X 0,Y 347.854,Z 440.156,A -85,B 0,C 180,E1 -13845.969,E2 -13845.969} C_VEL
LIN {X 0,Y 347.881,Z 440.227,A -85,B 0,C 180,E1 -13848.271,E2 -13848.271} C_VEL
LIN {X 0,Y 348.681,Z 443.105,A -85,B 0,C 180,E1 -13849.523,E2 -13849.523} C_VEL
LIN {X 0,Y 356.497,Z 456.997,A -85,B 0,C 180,E1 -13850.952,E2 -13850.952} C_VEL
LIN {X 0,Y 361.147,Z 467.09,A -85,B 0,C 180,E1 -13851.789,E2 -13851.789} C_VEL
LIN {X 0,Y 361.534,Z 468.138,A -85,B 0,C 180,E1 -13851.863,E2 -13851.863} C_VEL
LIN {X 0,Y 358.172,Z 547.065,A -85,B 0,C 180,E1 -13854.052,E2 -13854.052} C_VEL
LIN {X 0,Y 357.535,Z 560.3,A -85,B 0,C 180,E1 -13854.642,E2 -13854.642} C_VEL
LIN {X 0,Y 356.82,Z 571.506,A -85,B 0,C 180,E1 -13855.34,E2 -13855.34} C_VEL
LIN {X 0,Y 355.647,Z 583.665,A -85,B 0,C 180,E1 -13856.318,E2 -13856.318} C_VEL
LIN {X 0,Y 354.303,Z 595.786,A -85,B 0,C 180,E1 -13857.584,E2 -13857.584} C_VEL
LIN {X 0,Y 353.081,Z 605.511,A -85,B 0,C 180,E1 -13858.859,E2 -13858.859} C_VEL
LIN {X 0,Y 351.962,Z 613.868,A -85,B 0,C 180,E1 -13860.196,E2 -13860.196} C_VEL
LIN {X 0,Y 350.793,Z 621.714,A -85,B 0,C 180,E1 -13861.722,E2 -13861.722} C_VEL
LIN {X 0,Y 349.704,Z 628.908,A -85,B 0,C 180,E1 -13863.456,E2 -13863.456} C_VEL
LIN {X 0,Y 348.68,Z 635.216,A -85,B 0,C 180,E1 -13865.407,E2 -13865.407} C_VEL
LIN {X 0,Y 348.049,Z 639.131,A -85,B 0,C 180,E1 -13866.959,E2 -13866.959} C_VEL
LIN {X 0,Y 347.636,Z 641.471,A -85,B 0,C 180,E1 -13868.136,E2 -13868.136} C_VEL
LIN {X 0,Y 347.29,Z 643.368,A -85,B 0,C 180,E1 -13869.317,E2 -13869.317} C_VEL
LIN {X 0,Y 346.995,Z 644.815,A -85,B 0,C 180,E1 -13870.503,E2 -13870.503} C_VEL
LIN {X 0,Y 346.77,Z 645.774,A -85,B 0,C 180,E1 -13871.693,E2 -13871.693} C_VEL
LIN {X 0,Y 346.602,Z 646.398,A -85,B 0,C 180,E1 -13873.27,E2 -13873.27} C_VEL
LIN {X 0,Y 346.451,Z 646.033,A -85,B 0,C 180,E1 -13875.291,E2 -13875.291} C_VEL
LIN {X 0,Y 346.46,Z 645.213,A -85,B 0,C 180,E1 -13876.499,E2 -13876.499} C_VEL
LIN {X 0,Y 346.49,Z 643.946,A -85,B 0,C 180,E1 -13877.713,E2 -13877.713} C_VEL
LIN {X 0,Y 346.673,Z 641.096,A -85,B 0,C 180,E1 -13879.542,E2 -13879.542} C_VEL
LIN {X 0,Y 346.957,Z 637.051,A -85,B 0,C 180,E1 -13881.384,E2 -13881.384} C_VEL
LIN {X 0,Y 347.31,Z 631.662,A -85,B 0,C 180,E1 -13883.241,E2 -13883.241} C_VEL
LIN {X 0,Y 347.891,Z 624.76,A -85,B 0,C 180,E1 -13885.102,E2 -13885.102} C_VEL
LIN {X 0,Y 348.512,Z 617.577,A -85,B 0,C 180,E1 -13886.66,E2 -13886.66} C_VEL
LIN {X 0,Y 349.232,Z 608.718,A -85,B 0,C 180,E1 -13888.224,E2 -13888.224} C_VEL
LIN {X 0,Y 349.991,Z 598.93,A -85,B 0,C 180,E1 -13889.636,E2 -13889.636} C_VEL
LIN {X 0,Y 350.818,Z 588.711,A -85,B 0,C 180,E1 -13890.836,E2 -13890.836} C_VEL
LIN {X 0,Y 351.622,Z 576.408,A -85,B 0,C 180,E1 -13891.983,E2 -13891.983} C_VEL
LIN {X 0,Y 352.331,Z 563.895,A -85,B 0,C 180,E1 -13892.883,E2 -13892.883} C_VEL
LIN {X 0,Y 352.841,Z 551.08,A -85,B 0,C 180,E1 -13893.558,E2 -13893.558} C_VEL
LIN {X 0,Y 353.237,Z 536.928,A -85,B 0,C 180,E1 -13894.048,E2 -13894.048} C_VEL
LIN {X 0,Y 355.034,Z 460.682,A -85,B 0,C 180,E1 -13895.937,E2 -13895.937} C_VEL
LIN {X 0,Y 347.801,Z 440.16,A -85,B 0,C 180,E1 -13896.861,E2 -13896.861} C_VEL
LIN {X 0,Y 347.7,Z 440.176,A -85,B 0,C 180,E1 -13900.302,E2 -13900.302} C_VEL
LIN {X 0,Y 347.724,Z 440.167,A -85,B 0,C 180,E1 -13903.408,E2 -13903.408} C_VEL
LIN {X 0,Y 347.726,Z 440.171,A -85,B 0,C 180,E1 -13906.686,E2 -13906.686} C_VEL
LIN {X 0,Y 347.703,Z 440.174,A -85,B 0,C 180,E1 -13910.182,E2 -13910.182} C_VEL
LIN {X 0,Y 347.757,Z 440.167,A -85,B 0,C 180,E1 -13912.678,E2 -13912.678} C_VEL
LIN {X 0,Y 347.75,Z 440.166,A -85,B 0,C 180,E1 -13915.956,E2 -13915.956} C_VEL
LIN {X 0,Y 347.743,Z 440.165,A -85,B 0,C 180,E1 -13919.651,E2 -13919.651} C_VEL
LIN {X 0,Y 347.75,Z 440.164,A -85,B 0,C 180,E1 -13923.601,E2 -13923.601} C_VEL
LIN {X 0,Y 347.772,Z 440.165,A -85,B 0,C 180,E1 -13926.16,E2 -13926.16} C_VEL
LIN {X 0,Y 347.814,Z 440.158,A -85,B 0,C 180,E1 -13929.909,E2 -13929.909} C_VEL
LIN {X 0,Y 347.868,Z 440.155,A -85,B 0,C 180,E1 -13932.359,E2 -13932.359} C_VEL
LIN {X 0,Y 347.899,Z 440.147,A -85,B 0,C 180,E1 -13935.97,E2 -13935.97} C_VEL
LIN {X 0,Y 347.898,Z 440.146,A -85,B 0,C 180,E1 -13939.524,E2 -13939.524} C_VEL
LIN {X 0,Y 348.058,Z 440.127,A -85,B 0,C 180,E1 -13943.041,E2 -13943.041} C_VEL
LIN {X 0,Y 348.204,Z 440.108,A -85,B 0,C 180,E1 -13947.686,E2 -13947.686} C_VEL
LIN {X 0,Y 348.284,Z 440.099,A -85,B 0,C 180,E1 -13950,E2 -13950} C_VEL
LIN {X 0,Y 348.196,Z 440.113,A -85,B 0,C 180,E1 -13952.313,E2 -13952.313} C_VEL
LIN {X 0,Y 348.079,Z 440.125,A -85,B 0,C 180,E1 -13956.958,E2 -13956.958} C_VEL
LIN {X 0,Y 347.928,Z 440.148,A -85,B 0,C 180,E1 -13960.474,E2 -13960.474} C_VEL
LIN {X 0,Y 347.899,Z 440.148,A -85,B 0,C 180,E1 -13964.149,E2 -13964.149} C_VEL
LIN {X 0,Y 347.829,Z 440.158,A -85,B 0,C 180,E1 -13968.259,E2 -13968.259} C_VEL
LIN {X 0,Y 347.768,Z 440.162,A -85,B 0,C 180,E1 -13971.626,E2 -13971.626} C_VEL
LIN {X 0,Y 347.775,Z 440.162,A -85,B 0,C 180,E1 -13975.111,E2 -13975.111} C_VEL
LIN {X 0,Y 347.74,Z 440.165,A -85,B 0,C 180,E1 -13977.7,E2 -13977.7} C_VEL
LIN {X 0,Y 347.74,Z 440.17,A -85,B 0,C 180,E1 -13980.348,E2 -13980.348} C_VEL
LIN {X 0,Y 347.748,Z 440.166,A -85,B 0,C 180,E1 -13984.043,E2 -13984.043} C_VEL
LIN {X 0,Y 347.756,Z 440.164,A -85,B 0,C 180,E1 -13987.321,E2 -13987.321} C_VEL
LIN {X 0,Y 347.703,Z 440.169,A -85,B 0,C 180,E1 -13991.104,E2 -13991.104} C_VEL
LIN {X 0,Y 347.075,Z 440.251,A -85,B 0,C 180,E1 -13992.071,E2 -13992.071} C_VEL
LIN {X 0,Y 344.229,Z 440.609,A -85,B 0,C 180,E1 -13993.643,E2 -13993.643} C_VEL
LIN {X 0,Y 341.791,Z 440.914,A -85,B 0,C 180,E1 -13994.917,E2 -13994.917} C_VEL
LIN {X 0,Y 340.738,Z 441.042,A -85,B 0,C 180,E1 -13995.902,E2 -13995.902} C_VEL
LIN {X 0,Y 340.65,Z 441.051,A -85,B 0,C 180,E1 -13996.236,E2 -13996.236} C_VEL
LIN {X 0,Y 340.683,Z 441.045,A -85,B 0,C 180,E1 -13999.754,E2 -13999.754} C_VEL
LIN {X 0,Y 340.703,Z 441.043,A -85,B 0,C 180,E1 -14003.258,E2 -14003.258} C_VEL
LIN {X 0,Y 340.691,Z 441.046,A -85,B 0,C 180,E1 -14006.153,E2 -14006.153} C_VEL
LIN {X 0,Y 340.74,Z 441.041,A -85,B 0,C 180,E1 -14010.329,E2 -14010.329} C_VEL
LIN {X 0,Y 340.802,Z 441.032,A -85,B 0,C 180,E1 -14013.02,E2 -14013.02} C_VEL
LIN {X 0,Y 340.729,Z 441.042,A -85,B 0,C 180,E1 -14016.927,E2 -14016.927} C_VEL
LIN {X 0,Y 340.79,Z 441.036,A -85,B 0,C 180,E1 -14020.733,E2 -14020.733} C_VEL
LIN {X 0,Y 340.786,Z 441.033,A -85,B 0,C 180,E1 -14023.219,E2 -14023.219} C_VEL
LIN {X 0,Y 340.843,Z 441.028,A -85,B 0,C 180,E1 -14026.89,E2 -14026.89} C_VEL
LIN {X 0,Y 340.923,Z 441.02,A -85,B 0,C 180,E1 -14030.508,E2 -14030.508} C_VEL
LIN {X 0,Y 341.05,Z 441.002,A -85,B 0,C 180,E1 -14032.898,E2 -14032.898} C_VEL
LIN {X 0,Y 341.167,Z 440.984,A -85,B 0,C 180,E1 -14037.639,E2 -14037.639} C_VEL
LIN {X 0,Y 341.294,Z 440.969,A -85,B 0,C 180,E1 -14040,E2 -14040} C_VEL
LIN {X 0,Y 341.168,Z 440.987,A -85,B 0,C 180,E1 -14042.361,E2 -14042.361} C_VEL
LIN {X 0,Y 341.075,Z 440.998,A -85,B 0,C 180,E1 -14047.102,E2 -14047.102} C_VEL
LIN {X 0,Y 340.87,Z 441.027,A -85,B 0,C 180,E1 -14050.694,E2 -14050.694} C_VEL
LIN {X 0,Y 340.862,Z 441.025,A -85,B 0,C 180,E1 -14054.325,E2 -14054.325} C_VEL
LIN {X 0,Y 340.837,Z 441.029,A -85,B 0,C 180,E1 -14058.467,E2 -14058.467} C_VEL
LIN {X 0,Y 340.717,Z 441.04,A -85,B 0,C 180,E1 -14061.842,E2 -14061.842} C_VEL
LIN {X 0,Y 340.771,Z 441.033,A -85,B 0,C 180,E1 -14065.665,E2 -14065.665} C_VEL
LIN {X 0,Y 340.741,Z 441.04,A -85,B 0,C 180,E1 -14068.32,E2 -14068.32} C_VEL
LIN {X 0,Y 340.703,Z 441.045,A -85,B 0,C 180,E1 -14071.044,E2 -14071.044} C_VEL
LIN {X 0,Y 340.718,Z 441.041,A -85,B 0,C 180,E1 -14075.279,E2 -14075.279} C_VEL
LIN {X 0,Y 340.709,Z 441.044,A -85,B 0,C 180,E1 -14078.386,E2 -14078.386} C_VEL
LIN {X 0,Y 340.699,Z 441.043,A -85,B 0,C 180,E1 -14082.046,E2 -14082.046} C_VEL
LIN {X 0,Y 340.682,Z 441.045,A -85,B 0,C 180,E1 -14085.462,E2 -14085.462} C_VEL
LIN {X 0,Y 340.687,Z 441.05,A -85,B 0,C 180,E1 -14088.691,E2 -14088.691} C_VEL
LIN {X 0,Y 340.733,Z 441.038,A -85,B 0,C 180,E1 -14091.773,E2 -14091.773} C_VEL
LIN {X 0,Y 340.723,Z 441.042,A -85,B 0,C 180,E1 -14095.596,E2 -14095.596} C_VEL
LIN {X 0,Y 340.777,Z 441.229,A -85,B 0,C 180,E1 -14097.531,E2 -14097.531} C_VEL
LIN {X 0,Y 344.342,Z 458.012,A -85,B 0,C 180,E1 -14101.581,E2 -14101.581} C_VEL
LIN {X 0,Y 345.252,Z 462.991,A -85,B 0,C 180,E1 -14102.741,E2 -14102.741} C_VEL
LIN {X 0,Y 344.007,Z 476.054,A -85,B 0,C 180,E1 -14105.563,E2 -14105.563} C_VEL
LIN {X 0,Y 343.025,Z 486.07,A -85,B 0,C 180,E1 -14107.707,E2 -14107.707} C_VEL
LIN {X 0,Y 347.588,Z 527.623,A -85,B 0,C 180,E1 -14109.054,E2 -14109.054} C_VEL
LIN {X 0,Y 345.83,Z 596.169,A -85,B 0,C 180,E1 -14110.833,E2 -14110.833} C_VEL
LIN {X 0,Y 345.07,Z 610.28,A -85,B 0,C 180,E1 -14111.444,E2 -14111.444} C_VEL
LIN {X 0,Y 344.313,Z 621.946,A -85,B 0,C 180,E1 -14112.172,E2 -14112.172} C_VEL
LIN {X 0,Y 343.425,Z 632.751,A -85,B 0,C 180,E1 -14113.046,E2 -14113.046} C_VEL
LIN {X 0,Y 342.489,Z 644.248,A -85,B 0,C 180,E1 -14114.223,E2 -14114.223} C_VEL
LIN {X 0,Y 341.505,Z 654.632,A -85,B 0,C 180,E1 -14115.547,E2 -14115.547} C_VEL
LIN {X 0,Y 340.8,Z 663.208,A -85,B 0,C 180,E1 -14116.889,E2 -14116.889} C_VEL
LIN {X 0,Y 340.134,Z 672.486,A -85,B 0,C 180,E1 -14118.68,E2 -14118.68} C_VEL
LIN {X 0,Y 339.664,Z 679.933,A -85,B 0,C 180,E1 -14120.473,E2 -14120.473} C_VEL
LIN {X 0,Y 339.433,Z 685.824,A -85,B 0,C 180,E1 -14122.266,E2 -14122.266} C_VEL
LIN {X 0,Y 339.347,Z 690.401,A -85,B 0,C 180,E1 -14124.057,E2 -14124.057} C_VEL
LIN {X 0,Y 339.359,Z 692.786,A -85,B 0,C 180,E1 -14125.249,E2 -14125.249} C_VEL
LIN {X 0,Y 339.353,Z 694.701,A -85,B 0,C 180,E1 -14126.438,E2 -14126.438} C_VEL
LIN {X 0,Y 339.481,Z 696.125,A -85,B 0,C 180,E1 -14127.627,E2 -14127.627} C_VEL
LIN {X 0,Y 339.484,Z 697.078,A -85,B 0,C 180,E1 -14128.814,E2 -14128.814} C_VEL
LIN {X 0,Y 339.499,Z 697.606,A -85,B 0,C 180,E1 -14130,E2 -14130} C_VEL
LIN {X 0,Y 339.446,Z 697.689,A -85,B 0,C 180,E1 -14131.187,E2 -14131.187} C_VEL
LIN {X 0,Y 339.413,Z 697.3,A -85,B 0,C 180,E1 -14132.374,E2 -14132.374} C_VEL
LIN {X 0,Y 339.244,Z 696.48,A -85,B 0,C 180,E1 -14133.564,E2 -14133.564} C_VEL
LIN {X 0,Y 339.229,Z 695.249,A -85,B 0,C 180,E1 -14134.754,E2 -14134.754} C_VEL
LIN {X 0,Y 339.199,Z 692.531,A -85,B 0,C 180,E1 -14136.544,E2 -14136.544} C_VEL
LIN {X 0,Y 339.427,Z 688.765,A -85,B 0,C 180,E1 -14138.334,E2 -14138.334} C_VEL
LIN {X 0,Y 339.811,Z 683.89,A -85,B 0,C 180,E1 -14140.126,E2 -14140.126} C_VEL
LIN {X 0,Y 340.455,Z 677.766,A -85,B 0,C 180,E1 -14141.914,E2 -14141.914} C_VEL
LIN {X 0,Y 341.409,Z 670.149,A -85,B 0,C 180,E1 -14143.694,E2 -14143.694} C_VEL
LIN {X 0,Y 342.677,Z 660.755,A -85,B 0,C 180,E1 -14145.464,E2 -14145.464} C_VEL
LIN {X 0,Y 344.035,Z 651.191,A -85,B 0,C 180,E1 -14146.924,E2 -14146.924} C_VEL
LIN {X 0,Y 345.673,Z 639.439,A -85,B 0,C 180,E1 -14148.369,E2 -14148.369} C_VEL
LIN {X 0,Y 347.254,Z 627.761,A -85,B 0,C 180,E1 -14149.509,E2 -14149.509} C_VEL
LIN {X 0,Y 348.82,Z 614.578,A -85,B 0,C 180,E1 -14150.492,E2 -14150.492} C_VEL
LIN {X 0,Y 350.259,Z 600.632,A -85,B 0,C 180,E1 -14151.25,E2 -14151.25} C_VEL
LIN {X 0,Y 351.055,Z 586.482,A -85,B 0,C 180,E1 -14151.777,E2 -14151.777} C_VEL
LIN {X 0,Y 353.576,Z 527.75,A -85,B 0,C 180,E1 -14153.404,E2 -14153.404} C_VEL
LIN {X 0,Y 352.067,Z 511.489,A -85,B 0,C 180,E1 -14154.099,E2 -14154.099} C_VEL
LIN {X 0,Y 349.592,Z 495.784,A -85,B 0,C 180,E1 -14154.902,E2 -14154.902} C_VEL
LIN {X 0,Y 346.217,Z 479.231,A -85,B 0,C 180,E1 -14155.917,E2 -14155.917} C_VEL
LIN {X 0,Y 347.633,Z 470.316,A -85,B 0,C 180,E1 -14158.037,E2 -14158.037} C_VEL
LIN {X 0,Y 346.457,Z 462.862,A -85,B 0,C 180,E1 -14160.153,E2 -14160.153} C_VEL
LIN {X 0,Y 344.203,Z 453.416,A -85,B 0,C 180,E1 -14163.16,E2 -14163.16} C_VEL
LIN {X 0,Y 342.181,Z 445.98,A -85,B 0,C 180,E1 -14165.829,E2 -14165.829} C_VEL
LIN {X 0,Y 340.741,Z 441.042,A -85,B 0,C 180,E1 -14167.852,E2 -14167.852} C_VEL
LIN {X 0,Y 340.689,Z 441.049,A -85,B 0,C 180,E1 -14171.31,E2 -14171.31} C_VEL
LIN {X 0,Y 340.687,Z 441.049,A -85,B 0,C 180,E1 -14174.539,E2 -14174.539} C_VEL
LIN {X 0,Y 340.702,Z 441.045,A -85,B 0,C 180,E1 -14177.955,E2 -14177.955} C_VEL
LIN {X 0,Y 340.738,Z 441.039,A -85,B 0,C 180,E1 -14181.773,E2 -14181.773} C_VEL
LIN {X 0,Y 340.726,Z 441.038,A -85,B 0,C 180,E1 -14185.596,E2 -14185.596} C_VEL
LIN {X 0,Y 340.698,Z 441.045,A -85,B 0,C 180,E1 -14188.955,E2 -14188.955} C_VEL
LIN {X 0,Y 340.721,Z 441.044,A -85,B 0,C 180,E1 -14193.013,E2 -14193.013} C_VEL
LIN {X 0,Y 340.704,Z 441.046,A -85,B 0,C 180,E1 -14196.925,E2 -14196.925} C_VEL
LIN {X 0,Y 340.692,Z 441.047,A -85,B 0,C 180,E1 -14200.728,E2 -14200.728} C_VEL
LIN {X 0,Y 340.722,Z 441.043,A -85,B 0,C 180,E1 -14203.215,E2 -14203.215} C_VEL
LIN {X 0,Y 340.817,Z 441.032,A -85,B 0,C 180,E1 -14206.889,E2 -14206.889} C_VEL
LIN {X 0,Y 340.86,Z 441.27,A -85,B 0,C 180,E1 -14207.345,E2 -14207.345} C_VEL
LIN {X 0,Y 341.629,Z 444.009,A -85,B 0,C 180,E1 -14208.617,E2 -14208.617} C_VEL
LIN {X 0,Y 348.871,Z 456.365,A -85,B 0,C 180,E1 -14210.028,E2 -14210.028} C_VEL
LIN {X 0,Y 354.15,Z 466.9,A -85,B 0,C 180,E1 -14211.035,E2 -14211.035} C_VEL
LIN {X 0,Y 355.581,Z 470.533,A -85,B 0,C 180,E1 -14211.313,E2 -14211.313} C_VEL
LIN {X 0,Y 351.959,Z 547.857,A -85,B 0,C 180,E1 -14213.515,E2 -14213.515} C_VEL
LIN {X 0,Y 351.182,Z 562.218,A -85,B 0,C 180,E1 -14214.185,E2 -14214.185} C_VEL
LIN {X 0,Y 350.342,Z 574.048,A -85,B 0,C 180,E1 -14214.965,E2 -14214.965} C_VEL
LIN {X 0,Y 349.116,Z 585.776,A -85,B 0,C 180,E1 -14215.96,E2 -14215.96} C_VEL
LIN {X 0,Y 347.86,Z 596.421,A -85,B 0,C 180,E1 -14217.105,E2 -14217.105} C_VEL
LIN {X 0,Y 346.425,Z 607.074,A -85,B 0,C 180,E1 -14218.547,E2 -14218.547} C_VEL
LIN {X 0,Y 345.163,Z 615.735,A -85,B 0,C 180,E1 -14220,E2 -14220} C_VEL
LIN {X 0,Y 343.789,Z 624.25,A -85,B 0,C 180,E1 -14221.757,E2 -14221.757} C_VEL
LIN {X 0,Y 342.68,Z 631.037,A -85,B 0,C 180,E1 -14223.527,E2 -14223.527} C_VEL
LIN {X 0,Y 341.715,Z 636.455,A -85,B 0,C 180,E1 -14225.31,E2 -14225.31} C_VEL
LIN {X 0,Y 340.96,Z 640.65,A -85,B 0,C 180,E1 -14227.104,E2 -14227.104} C_VEL
LIN {X 0,Y 340.533,Z 642.85,A -85,B 0,C 180,E1 -14228.306,E2 -14228.306} C_VEL
LIN {X 0,Y 340.184,Z 644.547,A -85,B 0,C 180,E1 -14229.513,E2 -14229.513} C_VEL
LIN {X 0,Y 339.903,Z 645.791,A -85,B 0,C 180,E1 -14230.725,E2 -14230.725} C_VEL
LIN {X 0,Y 339.692,Z 646.616,A -85,B 0,C 180,E1 -14231.94,E2 -14231.94} C_VEL
LIN {X 0,Y 339.517,Z 646.99,A -85,B 0,C 180,E1 -14233.367,E2 -14233.367} C_VEL
LIN {X 0,Y 339.383,Z 646.37,A -85,B 0,C 180,E1 -14235.617,E2 -14235.617} C_VEL
LIN {X 0,Y 339.424,Z 644.382,A -85,B 0,C 180,E1 -14237.736,E2 -14237.736} C_VEL
LIN {X 0,Y 339.645,Z 640.759,A -85,B 0,C 180,E1 -14239.963,E2 -14239.963} C_VEL
LIN {X 0,Y 339.961,Z 636.404,A -85,B 0,C 180,E1 -14241.846,E2 -14241.846} C_VEL
LIN {X 0,Y 340.371,Z 630.66,A -85,B 0,C 180,E1 -14243.743,E2 -14243.743} C_VEL
LIN {X 0,Y 340.989,Z 623.26,A -85,B 0,C 180,E1 -14245.647,E2 -14245.647} C_VEL
LIN {X 0,Y 341.631,Z 615.766,A -85,B 0,C 180,E1 -14247.207,E2 -14247.207} C_VEL
LIN {X 0,Y 342.474,Z 606.207,A -85,B 0,C 180,E1 -14248.832,E2 -14248.832} C_VEL
LIN {X 0,Y 343.257,Z 595.635,A -85,B 0,C 180,E1 -14250.277,E2 -14250.277} C_VEL
LIN {X 0,Y 344.169,Z 584.51,A -85,B 0,C 180,E1 -14251.5,E2 -14251.5} C_VEL
LIN {X 0,Y 344.936,Z 572.955,A -85,B 0,C 180,E1 -14252.506,E2 -14252.506} C_VEL
LIN {X 0,Y 345.632,Z 559.884,A -85,B 0,C 180,E1 -14253.374,E2 -14253.374} C_VEL
LIN {X 0,Y 346.101,Z 547.306,A -85,B 0,C 180,E1 -14253.979,E2 -14253.979} C_VEL
LIN {X 0,Y 346.482,Z 530.063,A -85,B 0,C 180,E1 -14254.489,E2 -14254.489} C_VEL
LIN {X 0,Y 348.205,Z 462.213,A -85,B 0,C 180,E1 -14256.223,E2 -14256.223} C_VEL
LIN {X 0,Y 340.746,Z 441.037,A -85,B 0,C 180,E1 -14257.182,E2 -14257.182} C_VEL
LIN {X 0,Y 340.673,Z 441.046,A -85,B 0,C 180,E1 -14261.312,E2 -14261.312} C_VEL
LIN {X 0,Y 340.642,Z 441.054,A -85,B 0,C 180,E1 -14264.546,E2 -14264.546} C_VEL
LIN {X 0,Y 340.695,Z 441.045,A -85,B 0,C 180,E1 -14267.955,E2 -14267.955} C_VEL
LIN {X 0,Y 340.72,Z 441.041,A -85,B 0,C 180,E1 -14271.77,E2 -14271.77} C_VEL
LIN {X 0,Y 340.725,Z 441.039,A -85,B 0,C 180,E1 -14275.595,E2 -14275.595} C_VEL
LIN {X 0,Y 340.696,Z 441.044,A -85,B 0,C 180,E1 -14278.955,E2 -14278.955} C_VEL
LIN {X 0,Y 340.721,Z 441.041,A -85,B 0,C 180,E1 -14283.012,E2 -14283.012} C_VEL
LIN {X 0,Y 340.743,Z 441.037,A -85,B 0,C 180,E1 -14285.637,E2 -14285.637} C_VEL
LIN {X 0,Y 340.746,Z 441.037,A -85,B 0,C 180,E1 -14289.474,E2 -14289.474} C_VEL
LIN {X 0,Y 340.86,Z 441.024,A -85,B 0,C 180,E1 -14291.984,E2 -14291.984} C_VEL
LIN {X 0,Y 340.871,Z 441.021,A -85,B 0,C 180,E1 -14295.705,E2 -14295.705} C_VEL
LIN {X 0,Y 340.85,Z 441.024,A -85,B 0,C 180,E1 -14299.305,E2 -14299.305} C_VEL
LIN {X 0,Y 341.004,Z 441.007,A -85,B 0,C 180,E1 -14302.896,E2 -14302.896} C_VEL
LIN {X 0,Y 340.829,Z 441.027,A -85,B 0,C 180,E1 -14305.268,E2 -14305.268} C_VEL
LIN {X 0,Y 341.165,Z 440.985,A -85,B 0,C 180,E1 -14307.638,E2 -14307.638} C_VEL
LIN {X 0,Y 341.236,Z 440.977,A -85,B 0,C 180,E1 -14310,E2 -14310} C_VEL
LIN {X 0,Y 341.157,Z 440.99,A -85,B 0,C 180,E1 -14312.361,E2 -14312.361} C_VEL
LIN {X 0,Y 341.047,Z 441,A -85,B 0,C 180,E1 -14317.102,E2 -14317.102} C_VEL
LIN {X 0,Y 340.87,Z 441.025,A -85,B 0,C 180,E1 -14320.693,E2 -14320.693} C_VEL
LIN {X 0,Y 340.864,Z 441.026,A -85,B 0,C 180,E1 -14324.324,E2 -14324.324} C_VEL
LIN {X 0,Y 340.786,Z 441.037,A -85,B 0,C 180,E1 -14328.44,E2 -14328.44} C_VEL
LIN {X 0,Y 340.718,Z 441.041,A -85,B 0,C 180,E1 -14331.841,E2 -14331.841} C_VEL
LIN {X 0,Y 340.727,Z 441.039,A -85,B 0,C 180,E1 -14335.668,E2 -14335.668} C_VEL
LIN {X 0,Y 340.707,Z 441.042,A -85,B 0,C 180,E1 -14339.674,E2 -14339.674} C_VEL
LIN {X 0,Y 340.685,Z 441.049,A -85,B 0,C 180,E1 -14342.435,E2 -14342.435} C_VEL
LIN {X 0,Y 340.717,Z 441.041,A -85,B 0,C 180,E1 -14345.279,E2 -14345.279} C_VEL
LIN {X 0,Y 340.693,Z 441.048,A -85,B 0,C 180,E1 -14348.382,E2 -14348.382} C_VEL
LIN {X 0,Y 340.693,Z 441.045,A -85,B 0,C 180,E1 -14352.044,E2 -14352.044} C_VEL
LIN {X 0,Y 340.65,Z 441.051,A -85,B 0,C 180,E1 -14356.236,E2 -14356.236} C_VEL
LIN {X 0,Y 339.986,Z 441.133,A -85,B 0,C 180,E1 -14357.223,E2 -14357.223} C_VEL
LIN {X 0,Y 337.163,Z 441.487,A -85,B 0,C 180,E1 -14358.829,E2 -14358.829} C_VEL
LIN {X 0,Y 334.766,Z 441.784,A -85,B 0,C 180,E1 -14360.129,E2 -14360.129} C_VEL
LIN {X 0,Y 333.728,Z 441.913,A -85,B 0,C 180,E1 -14361.135,E2 -14361.135} C_VEL
LIN {X 0,Y 333.638,Z 441.922,A -85,B 0,C 180,E1 -14361.476,E2 -14361.476} C_VEL
LIN {X 0,Y 333.673,Z 441.918,A -85,B 0,C 180,E1 -14365.341,E2 -14365.341} C_VEL
LIN {X 0,Y 333.689,Z 441.916,A -85,B 0,C 180,E1 -14369.637,E2 -14369.637} C_VEL
LIN {X 0,Y 333.739,Z 441.914,A -85,B 0,C 180,E1 -14372.401,E2 -14372.401} C_VEL
LIN {X 0,Y 333.725,Z 441.913,A -85,B 0,C 180,E1 -14375.091,E2 -14375.091} C_VEL
LIN {X 0,Y 333.684,Z 441.919,A -85,B 0,C 180,E1 -14379.019,E2 -14379.019} C_VEL
LIN {X 0,Y 333.793,Z 441.903,A -85,B 0,C 180,E1 -14381.589,E2 -14381.589} C_VEL
LIN {X 0,Y 333.807,Z 441.901,A -85,B 0,C 180,E1 -14385.577,E2 -14385.577} C_VEL
LIN {X 0,Y 333.833,Z 441.9,A -85,B 0,C 180,E1 -14389.078,E2 -14389.078} C_VEL
LIN {X 0,Y 334.004,Z 441.882,A -85,B 0,C 180,E1 -14392.747,E2 -14392.747} C_VEL
LIN {X 0,Y 333.803,Z 441.903,A -85,B 0,C 180,E1 -14395.169,E2 -14395.169} C_VEL
LIN {X 0,Y 334.104,Z 441.864,A -85,B 0,C 180,E1 -14397.589,E2 -14397.589} C_VEL
LIN {X 0,Y 334.245,Z 441.847,A -85,B 0,C 180,E1 -14400,E2 -14400} C_VEL
LIN {X 0,Y 334.105,Z 441.868,A -85,B 0,C 180,E1 -14402.411,E2 -14402.411} C_VEL
LIN {X 0,Y 334.025,Z 441.875,A -85,B 0,C 180,E1 -14407.253,E2 -14407.253} C_VEL
LIN {X 0,Y 333.833,Z 441.901,A -85,B 0,C 180,E1 -14410.922,E2 -14410.922} C_VEL
LIN {X 0,Y 333.808,Z 441.907,A -85,B 0,C 180,E1 -14414.634,E2 -14414.634} C_VEL
LIN {X 0,Y 333.796,Z 441.908,A -85,B 0,C 180,E1 -14418.656,E2 -14418.656} C_VEL
LIN {X 0,Y 333.656,Z 441.922,A -85,B 0,C 180,E1 -14422.281,E2 -14422.281} C_VEL
LIN {X 0,Y 333.735,Z 441.912,A -85,B 0,C 180,E1 -14426.247,E2 -14426.247} C_VEL
LIN {X 0,Y 333.71,Z 441.917,A -85,B 0,C 180,E1 -14428.972,E2 -14428.972} C_VEL
LIN {X 0,Y 333.643,Z 441.926,A -85,B 0,C 180,E1 -14432.587,E2 -14432.587} C_VEL
LIN {X 0,Y 333.676,Z 441.919,A -85,B 0,C 180,E1 -14436.139,E2 -14436.139} C_VEL
LIN {X 0,Y 333.646,Z 441.923,A -85,B 0,C 180,E1 -14439.193,E2 -14439.193} C_VEL
LIN {X 0,Y 333.633,Z 441.926,A -85,B 0,C 180,E1 -14442.501,E2 -14442.501} C_VEL
LIN {X 0,Y 333.62,Z 441.925,A -85,B 0,C 180,E1 -14445.959,E2 -14445.959} C_VEL
LIN {X 0,Y 333.647,Z 441.922,A -85,B 0,C 180,E1 -14449.316,E2 -14449.316} C_VEL
LIN {X 0,Y 333.665,Z 441.921,A -85,B 0,C 180,E1 -14453.168,E2 -14453.168} C_VEL
LIN {X 0,Y 333.673,Z 441.924,A -85,B 0,C 180,E1 -14456.796,E2 -14456.796} C_VEL
LIN {X 0,Y 333.713,Z 442.054,A -85,B 0,C 180,E1 -14457.243,E2 -14457.243} C_VEL
LIN {X 0,Y 337.295,Z 458.76,A -85,B 0,C 180,E1 -14461.365,E2 -14461.365} C_VEL
LIN {X 0,Y 338.255,Z 464.838,A -85,B 0,C 180,E1 -14462.8,E2 -14462.8} C_VEL
LIN {X 0,Y 336.419,Z 482.197,A -85,B 0,C 180,E1 -14466.615,E2 -14466.615} C_VEL
LIN {X 0,Y 336.096,Z 485.577,A -85,B 0,C 180,E1 -14467.355,E2 -14467.355} C_VEL
LIN {X 0,Y 340.731,Z 527.969,A -85,B 0,C 180,E1 -14468.766,E2 -14468.766} C_VEL
LIN {X 0,Y 338.895,Z 595.717,A -85,B 0,C 180,E1 -14470.583,E2 -14470.583} C_VEL
LIN {X 0,Y 338.145,Z 609.021,A -85,B 0,C 180,E1 -14471.168,E2 -14471.168} C_VEL
LIN {X 0,Y 337.363,Z 621.396,A -85,B 0,C 180,E1 -14471.949,E2 -14471.949} C_VEL
LIN {X 0,Y 336.447,Z 632.186,A -85,B 0,C 180,E1 -14472.84,E2 -14472.84} C_VEL
LIN {X 0,Y 335.474,Z 643.675,A -85,B 0,C 180,E1 -14474.041,E2 -14474.041} C_VEL
LIN {X 0,Y 334.466,Z 654.094,A -85,B 0,C 180,E1 -14475.396,E2 -14475.396} C_VEL
LIN {X 0,Y 333.85,Z 661.772,A -85,B 0,C 180,E1 -14476.611,E2 -14476.611} C_VEL
LIN {X 0,Y 333.246,Z 669.839,A -85,B 0,C 180,E1 -14478.134,E2 -14478.134} C_VEL
LIN {X 0,Y 332.682,Z 677.661,A -85,B 0,C 180,E1 -14479.963,E2 -14479.963} C_VEL
LIN {X 0,Y 332.431,Z 682.986,A -85,B 0,C 180,E1 -14481.49,E2 -14481.49} C_VEL
LIN {X 0,Y 332.301,Z 688.096,A -85,B 0,C 180,E1 -14483.321,E2 -14483.321} C_VEL
LIN {X 0,Y 332.302,Z 691.974,A -85,B 0,C 180,E1 -14485.148,E2 -14485.148} C_VEL
LIN {X 0,Y 332.276,Z 693.93,A -85,B 0,C 180,E1 -14486.362,E2 -14486.362} C_VEL
LIN {X 0,Y 332.418,Z 695.433,A -85,B 0,C 180,E1 -14487.577,E2 -14487.577} C_VEL
LIN {X 0,Y 332.419,Z 696.426,A -85,B 0,C 180,E1 -14488.789,E2 -14488.789} C_VEL
LIN {X 0,Y 332.43,Z 696.988,A -85,B 0,C 180,E1 -14490,E2 -14490} C_VEL
LIN {X 0,Y 332.382,Z 697.119,A -85,B 0,C 180,E1 -14491.212,E2 -14491.212} C_VEL
LIN {X 0,Y 332.314,Z 696.782,A -85,B 0,C 180,E1 -14492.425,E2 -14492.425} C_VEL
LIN {X 0,Y 332.16,Z 695.991,A -85,B 0,C 180,E1 -14493.64,E2 -14493.64} C_VEL
LIN {X 0,Y 332.139,Z 694.79,A -85,B 0,C 180,E1 -14494.856,E2 -14494.856} C_VEL
LIN {X 0,Y 332.119,Z 692.149,A -85,B 0,C 180,E1 -14496.684,E2 -14496.684} C_VEL
LIN {X 0,Y 332.352,Z 688.471,A -85,B 0,C 180,E1 -14498.513,E2 -14498.513} C_VEL
LIN {X 0,Y 332.775,Z 683.668,A -85,B 0,C 180,E1 -14500.342,E2 -14500.342} C_VEL
LIN {X 0,Y 333.496,Z 677.626,A -85,B 0,C 180,E1 -14502.166,E2 -14502.166} C_VEL
LIN {X 0,Y 334.484,Z 670.136,A -85,B 0,C 180,E1 -14503.983,E2 -14503.983} C_VEL
LIN {X 0,Y 335.828,Z 660.92,A -85,B 0,C 180,E1 -14505.787,E2 -14505.787} C_VEL
LIN {X 0,Y 337.451,Z 650.55,A -85,B 0,C 180,E1 -14507.421,E2 -14507.421} C_VEL
LIN {X 0,Y 338.985,Z 640.086,A -85,B 0,C 180,E1 -14508.745,E2 -14508.745} C_VEL
LIN {X 0,Y 340.869,Z 627.083,A -85,B 0,C 180,E1 -14510.046,E2 -14510.046} C_VEL
LIN {X 0,Y 342.497,Z 613.907,A -85,B 0,C 180,E1 -14511.045,E2 -14511.045} C_VEL
LIN {X 0,Y 344.044,Z 600.15,A -85,B 0,C 180,E1 -14511.81,E2 -14511.81} C_VEL
LIN {X 0,Y 344.918,Z 585.293,A -85,B 0,C 180,E1 -14512.382,E2 -14512.382} C_VEL
LIN {X 0,Y 347.526,Z 528.53,A -85,B 0,C 180,E1 -14513.997,E2 -14513.997} C_VEL
LIN {X 0,Y 346.137,Z 513.078,A -85,B 0,C 180,E1 -14514.683,E2 -14514.683} C_VEL
LIN {X 0,Y 343.742,Z 497.207,A -85,B 0,C 180,E1 -14515.535,E2 -14515.535} C_VEL
LIN {X 0,Y 340.431,Z 481.474,A -85,B 0,C 180,E1 -14516.53,E2 -14516.53} C_VEL
LIN {X 0,Y 339.834,Z 478.447,A -85,B 0,C 180,E1 -14516.744,E2 -14516.744} C_VEL
LIN {X 0,Y 340.924,Z 472.108,A -85,B 0,C 180,E1 -14518.304,E2 -14518.304} C_VEL
LIN {X 0,Y 339.755,Z 464.804,A -85,B 0,C 180,E1 -14520.45,E2 -14520.45} C_VEL
LIN {X 0,Y 337.529,Z 455.255,A -85,B 0,C 180,E1 -14523.604,E2 -14523.604} C_VEL
LIN {X 0,Y 335.531,Z 448.101,A -85,B 0,C 180,E1 -14526.3,E2 -14526.3} C_VEL
LIN {X 0,Y 333.66,Z 441.923,A -85,B 0,C 180,E1 -14529.005,E2 -14529.005} C_VEL
LIN {X 0,Y 333.637,Z 441.926,A -85,B 0,C 180,E1 -14532.5,E2 -14532.5} C_VEL
LIN {X 0,Y 333.623,Z 441.926,A -85,B 0,C 180,E1 -14535.959,E2 -14535.959} C_VEL
LIN {X 0,Y 333.65,Z 441.921,A -85,B 0,C 180,E1 -14539.316,E2 -14539.316} C_VEL
LIN {X 0,Y 333.67,Z 441.918,A -85,B 0,C 180,E1 -14543.168,E2 -14543.168} C_VEL
LIN {X 0,Y 333.64,Z 441.924,A -85,B 0,C 180,E1 -14546.792,E2 -14546.792} C_VEL
LIN {X 0,Y 333.665,Z 441.918,A -85,B 0,C 180,E1 -14549.723,E2 -14549.723} C_VEL
LIN {X 0,Y 333.67,Z 441.921,A -85,B 0,C 180,E1 -14552.394,E2 -14552.394} C_VEL
LIN {X 0,Y 333.645,Z 441.925,A -85,B 0,C 180,E1 -14556.408,E2 -14556.408} C_VEL
LIN {X 0,Y 333.642,Z 441.925,A -85,B 0,C 180,E1 -14559.017,E2 -14559.017} C_VEL
LIN {X 0,Y 333.708,Z 441.916,A -85,B 0,C 180,E1 -14561.584,E2 -14561.584} C_VEL
LIN {X 0,Y 333.782,Z 441.931,A -85,B 0,C 180,E1 -14566.11,E2 -14566.11} C_VEL
LIN {X 0,Y 334.644,Z 445.022,A -85,B 0,C 180,E1 -14567.646,E2 -14567.646} C_VEL
LIN {X 0,Y 336.997,Z 448.727,A -85,B 0,C 180,E1 -14568.149,E2 -14568.149} C_VEL
LIN {X 0,Y 345.012,Z 462.591,A -85,B 0,C 180,E1 -14569.784,E2 -14569.784} C_VEL
LIN {X 0,Y 349.577,Z 472.172,A -85,B 0,C 180,E1 -14570.69,E2 -14570.69} C_VEL
LIN {X 0,Y 345.802,Z 549.11,A -85,B 0,C 180,E1 -14572.959,E2 -14572.959} C_VEL
LIN {X 0,Y 344.986,Z 563.253,A -85,B 0,C 180,E1 -14573.64,E2 -14573.64} C_VEL
LIN {X 0,Y 344.087,Z 574.869,A -85,B 0,C 180,E1 -14574.432,E2 -14574.432} C_VEL
LIN {X 0,Y 342.783,Z 586.477,A -85,B 0,C 180,E1 -14575.443,E2 -14575.443} C_VEL
LIN {X 0,Y 341.454,Z 597.049,A -85,B 0,C 180,E1 -14576.607,E2 -14576.607} C_VEL
LIN {X 0,Y 340.045,Z 606.793,A -85,B 0,C 180,E1 -14577.927,E2 -14577.927} C_VEL
LIN {X 0,Y 338.672,Z 615.622,A -85,B 0,C 180,E1 -14579.405,E2 -14579.405} C_VEL
LIN {X 0,Y 337.223,Z 624.259,A -85,B 0,C 180,E1 -14581.194,E2 -14581.194} C_VEL
LIN {X 0,Y 335.997,Z 631.167,A -85,B 0,C 180,E1 -14582.997,E2 -14582.997} C_VEL
LIN {X 0,Y 334.927,Z 636.657,A -85,B 0,C 180,E1 -14584.815,E2 -14584.815} C_VEL
LIN {X 0,Y 334.102,Z 640.95,A -85,B 0,C 180,E1 -14586.644,E2 -14586.644} C_VEL
LIN {X 0,Y 333.444,Z 644.129,A -85,B 0,C 180,E1 -14588.484,E2 -14588.484} C_VEL
LIN {X 0,Y 333.075,Z 645.672,A -85,B 0,C 180,E1 -14589.718,E2 -14589.718} C_VEL
LIN {X 0,Y 332.803,Z 646.772,A -85,B 0,C 180,E1 -14590.956,E2 -14590.956} C_VEL
LIN {X 0,Y 332.591,Z 647.39,A -85,B 0,C 180,E1 -14592.199,E2 -14592.199} C_VEL
LIN {X 0,Y 332.443,Z 647.586,A -85,B 0,C 180,E1 -14593.475,E2 -14593.475} C_VEL
LIN {X 0,Y 332.326,Z 647.352,A -85,B 0,C 180,E1 -14594.701,E2 -14594.701} C_VEL
LIN {X 0,Y 332.288,Z 646.622,A -85,B 0,C 180,E1 -14595.959,E2 -14595.959} C_VEL
LIN {X 0,Y 332.35,Z 644.624,A -85,B 0,C 180,E1 -14597.899,E2 -14597.899} C_VEL
LIN {X 0,Y 332.541,Z 641.634,A -85,B 0,C 180,E1 -14599.764,E2 -14599.764} C_VEL
LIN {X 0,Y 332.837,Z 637.317,A -85,B 0,C 180,E1 -14601.707,E2 -14601.707} C_VEL
LIN {X 0,Y 333.237,Z 631.738,A -85,B 0,C 180,E1 -14603.623,E2 -14603.623} C_VEL
LIN {X 0,Y 333.861,Z 624.613,A -85,B 0,C 180,E1 -14605.534,E2 -14605.534} C_VEL
LIN {X 0,Y 334.53,Z 616.948,A -85,B 0,C 180,E1 -14607.19,E2 -14607.19} C_VEL
LIN {X 0,Y 335.385,Z 607.736,A -85,B 0,C 180,E1 -14608.814,E2 -14608.814} C_VEL
LIN {X 0,Y 336.146,Z 597.464,A -85,B 0,C 180,E1 -14610.283,E2 -14610.283} C_VEL
LIN {X 0,Y 337.107,Z 586.053,A -85,B 0,C 180,E1 -14611.588,E2 -14611.588} C_VEL
LIN {X 0,Y 337.896,Z 574.416,A -85,B 0,C 180,E1 -14612.648,E2 -14612.648} C_VEL
LIN {X 0,Y 338.633,Z 561.454,A -85,B 0,C 180,E1 -14613.544,E2 -14613.544} C_VEL
LIN {X 0,Y 339.16,Z 548.415,A -85,B 0,C 180,E1 -14614.2,E2 -14614.2} C_VEL
LIN {X 0,Y 339.515,Z 532.466,A -85,B 0,C 180,E1 -14614.698,E2 -14614.698} C_VEL
LIN {X 0,Y 341.306,Z 463.51,A -85,B 0,C 180,E1 -14616.513,E2 -14616.513} C_VEL
LIN {X 0,Y 333.692,Z 441.915,A -85,B 0,C 180,E1 -14617.516,E2 -14617.516} C_VEL
LIN {X 0,Y 333.606,Z 441.929,A -85,B 0,C 180,E1 -14620.774,E2 -14620.774} C_VEL
LIN {X 0,Y 333.594,Z 441.932,A -85,B 0,C 180,E1 -14624.25,E2 -14624.25} C_VEL
LIN {X 0,Y 333.64,Z 441.922,A -85,B 0,C 180,E1 -14627.617,E2 -14627.617} C_VEL
LIN {X 0,Y 333.618,Z 441.925,A -85,B 0,C 180,E1 -14631.21,E2 -14631.21} C_VEL
LIN {X 0,Y 333.677,Z 441.919,A -85,B 0,C 180,E1 -14633.86,E2 -14633.86} C_VEL
LIN {X 0,Y 333.646,Z 441.921,A -85,B 0,C 180,E1 -14637.413,E2 -14637.413} C_VEL
LIN {X 0,Y 333.656,Z 441.921,A -85,B 0,C 180,E1 -14641.022,E2 -14641.022} C_VEL
LIN {X 0,Y 333.698,Z 441.915,A -85,B 0,C 180,E1 -14645.088,E2 -14645.088} C_VEL
LIN {X 0,Y 333.682,Z 441.918,A -85,B 0,C 180,E1 -14649.019,E2 -14649.019} C_VEL
LIN {X 0,Y 333.796,Z 441.903,A -85,B 0,C 180,E1 -14651.589,E2 -14651.589} C_VEL
LIN {X 0,Y 333.81,Z 441.901,A -85,B 0,C 180,E1 -14655.576,E2 -14655.576} C_VEL
LIN {X 0,Y 333.819,Z 441.9,A -85,B 0,C 180,E1 -14659.077,E2 -14659.077} C_VEL
LIN {X 0,Y 333.959,Z 441.885,A -85,B 0,C 180,E1 -14662.746,E2 -14662.746} C_VEL
LIN {X 0,Y 333.794,Z 441.903,A -85,B 0,C 180,E1 -14665.168,E2 -14665.168} C_VEL
LIN {X 0,Y 334.102,Z 441.864,A -85,B 0,C 180,E1 -14667.588,E2 -14667.588} C_VEL
LIN {X 0,Y 334.189,Z 441.855,A -85,B 0,C 180,E1 -14670,E2 -14670} C_VEL
LIN {X 0,Y 334.094,Z 441.871,A -85,B 0,C 180,E1 -14672.411,E2 -14672.411} C_VEL
LIN {X 0,Y 334.009,Z 441.878,A -85,B 0,C 180,E1 -14676.039,E2 -14676.039} C_VEL
LIN {X 0,Y 333.849,Z 441.896,A -85,B 0,C 180,E1 -14679.695,E2 -14679.695} C_VEL
LIN {X 0,Y 333.797,Z 441.902,A -85,B 0,C 180,E1 -14683.391,E2 -14683.391} C_VEL
LIN {X 0,Y 333.719,Z 441.913,A -85,B 0,C 180,E1 -14687.147,E2 -14687.147} C_VEL
LIN {X 0,Y 333.686,Z 441.916,A -85,B 0,C 180,E1 -14689.693,E2 -14689.693} C_VEL
LIN {X 0,Y 333.667,Z 441.919,A -85,B 0,C 180,E1 -14693.59,E2 -14693.59} C_VEL
LIN {X 0,Y 333.662,Z 441.922,A -85,B 0,C 180,E1 -14696.252,E2 -14696.252} C_VEL
LIN {X 0,Y 333.661,Z 441.923,A -85,B 0,C 180,E1 -14700.277,E2 -14700.277} C_VEL
LIN {X 0,Y 333.636,Z 441.923,A -85,B 0,C 180,E1 -14703.208,E2 -14703.208} C_VEL
LIN {X 0,Y 333.674,Z 441.92,A -85,B 0,C 180,E1 -14706.139,E2 -14706.139} C_VEL
LIN {X 0,Y 333.619,Z 441.925,A -85,B 0,C 180,E1 -14709.196,E2 -14709.196} C_VEL
LIN {X 0,Y 333.628,Z 441.929,A -85,B 0,C 180,E1 -14712.499,E2 -14712.499} C_VEL
LIN {X 0,Y 333.583,Z 441.927,A -85,B 0,C 180,E1 -14716.231,E2 -14716.231} C_VEL
LIN {X 0,Y 333.644,Z 441.922,A -85,B 0,C 180,E1 -14719.315,E2 -14719.315} C_VEL
LIN {X 0,Y 333.638,Z 441.922,A -85,B 0,C 180,E1 -14721.476,E2 -14721.476} C_VEL
LIN {X 0,Y 332.952,Z 442.013,A -85,B 0,C 180,E1 -14722.484,E2 -14722.484} C_VEL
LIN {X 0,Y 330.082,Z 442.367,A -85,B 0,C 180,E1 -14724.125,E2 -14724.125} C_VEL
LIN {X 0,Y 327.678,Z 442.665,A -85,B 0,C 180,E1 -14725.453,E2 -14725.453} C_VEL
LIN {X 0,Y 326.673,Z 442.795,A -85,B 0,C 180,E1 -14726.482,E2 -14726.482} C_VEL
LIN {X 0,Y 326.604,Z 442.799,A -85,B 0,C 180,E1 -14726.83,E2 -14726.83} C_VEL
LIN {X 0,Y 326.647,Z 442.796,A -85,B 0,C 180,E1 -14730.34,E2 -14730.34} C_VEL
LIN {X 0,Y 326.689,Z 442.793,A -85,B 0,C 180,E1 -14734.516,E2 -14734.516} C_VEL
LIN {X 0,Y 326.647,Z 442.798,A -85,B 0,C 180,E1 -14738.545,E2 -14738.545} C_VEL
LIN {X 0,Y 326.743,Z 442.782,A -85,B 0,C 180,E1 -14741.177,E2 -14741.177} C_VEL
LIN {X 0,Y 326.762,Z 442.779,A -85,B 0,C 180,E1 -14745.433,E2 -14745.433} C_VEL
LIN {X 0,Y 326.769,Z 442.782,A -85,B 0,C 180,E1 -14748.839,E2 -14748.839} C_VEL
LIN {X 0,Y 326.959,Z 442.76,A -85,B 0,C 180,E1 -14752.59,E2 -14752.59} C_VEL
LIN {X 0,Y 326.77,Z 442.78,A -85,B 0,C 180,E1 -14755.065,E2 -14755.065} C_VEL
LIN {X 0,Y 327.045,Z 442.744,A -85,B 0,C 180,E1 -14757.537,E2 -14757.537} C_VEL
LIN {X 0,Y 327.197,Z 442.725,A -85,B 0,C 180,E1 -14760,E2 -14760} C_VEL
LIN {X 0,Y 327.046,Z 442.747,A -85,B 0,C 180,E1 -14762.463,E2 -14762.463} C_VEL
LIN {X 0,Y 326.996,Z 442.751,A -85,B 0,C 180,E1 -14766.169,E2 -14766.169} C_VEL
LIN {X 0,Y 326.914,Z 442.766,A -85,B 0,C 180,E1 -14768.655,E2 -14768.655} C_VEL
LIN {X 0,Y 326.734,Z 442.786,A -85,B 0,C 180,E1 -14772.421,E2 -14772.421} C_VEL
LIN {X 0,Y 326.754,Z 442.783,A -85,B 0,C 180,E1 -14774.958,E2 -14774.958} C_VEL
LIN {X 0,Y 326.732,Z 442.787,A -85,B 0,C 180,E1 -14778.838,E2 -14778.838} C_VEL
LIN {X 0,Y 326.602,Z 442.804,A -85,B 0,C 180,E1 -14782.789,E2 -14782.789} C_VEL
LIN {X 0,Y 326.689,Z 442.788,A -85,B 0,C 180,E1 -14785.484,E2 -14785.484} C_VEL
LIN {X 0,Y 326.66,Z 442.791,A -85,B 0,C 180,E1 -14789.659,E2 -14789.659} C_VEL
LIN {X 0,Y 326.606,Z 442.799,A -85,B 0,C 180,E1 -14794.02,E2 -14794.02} C_VEL
LIN {X 0,Y 326.627,Z 442.797,A -85,B 0,C 180,E1 -14797.239,E2 -14797.239} C_VEL
LIN {X 0,Y 326.577,Z 442.804,A -85,B 0,C 180,E1 -14801.132,E2 -14801.132} C_VEL
LIN {X 0,Y 326.557,Z 442.81,A -85,B 0,C 180,E1 -14804.748,E2 -14804.748} C_VEL
LIN {X 0,Y 326.576,Z 442.803,A -85,B 0,C 180,E1 -14808.155,E2 -14808.155} C_VEL
LIN {X 0,Y 326.598,Z 442.8,A -85,B 0,C 180,E1 -14811.388,E2 -14811.388} C_VEL
LIN {X 0,Y 326.62,Z 442.802,A -85,B 0,C 180,E1 -14814.852,E2 -14814.852} C_VEL
LIN {X 0,Y 326.663,Z 442.844,A -85,B 0,C 180,E1 -14816.945,E2 -14816.945} C_VEL
LIN {X 0,Y 330.095,Z 459.039,A -85,B 0,C 180,E1 -14821.031,E2 -14821.031} C_VEL
LIN {X 0,Y 331.211,Z 464.8,A -85,B 0,C 180,E1 -14822.436,E2 -14822.436} C_VEL
LIN {X 0,Y 330.338,Z 473.857,A -85,B 0,C 180,E1 -14824.481,E2 -14824.481} C_VEL
LIN {X 0,Y 329.174,Z 485.079,A -85,B 0,C 180,E1 -14826.992,E2 -14826.992} C_VEL
LIN {X 0,Y 333.77,Z 529.176,A -85,B 0,C 180,E1 -14828.505,E2 -14828.505} C_VEL
LIN {X 0,Y 331.972,Z 595.105,A -85,B 0,C 180,E1 -14830.322,E2 -14830.322} C_VEL
LIN {X 0,Y 331.208,Z 608.399,A -85,B 0,C 180,E1 -14830.919,E2 -14830.919} C_VEL
LIN {X 0,Y 330.394,Z 620.79,A -85,B 0,C 180,E1 -14831.715,E2 -14831.715} C_VEL
LIN {X 0,Y 329.472,Z 631.596,A -85,B 0,C 180,E1 -14832.625,E2 -14832.625} C_VEL
LIN {X 0,Y 328.468,Z 643.094,A -85,B 0,C 180,E1 -14833.85,E2 -14833.85} C_VEL
LIN {X 0,Y 327.429,Z 653.523,A -85,B 0,C 180,E1 -14835.234,E2 -14835.234} C_VEL
LIN {X 0,Y 326.718,Z 662.096,A -85,B 0,C 180,E1 -14836.63,E2 -14836.63} C_VEL
LIN {X 0,Y 326.016,Z 671.392,A -85,B 0,C 180,E1 -14838.498,E2 -14838.498} C_VEL
LIN {X 0,Y 325.522,Z 678.851,A -85,B 0,C 180,E1 -14840.368,E2 -14840.368} C_VEL
LIN {X 0,Y 325.31,Z 683.853,A -85,B 0,C 180,E1 -14841.928,E2 -14841.928} C_VEL
LIN {X 0,Y 325.233,Z 688.66,A -85,B 0,C 180,E1 -14843.798,E2 -14843.798} C_VEL
LIN {X 0,Y 325.245,Z 691.163,A -85,B 0,C 180,E1 -14845.042,E2 -14845.042} C_VEL
LIN {X 0,Y 325.2,Z 693.159,A -85,B 0,C 180,E1 -14846.283,E2 -14846.283} C_VEL
LIN {X 0,Y 325.356,Z 694.722,A -85,B 0,C 180,E1 -14847.524,E2 -14847.524} C_VEL
LIN {X 0,Y 325.356,Z 695.773,A -85,B 0,C 180,E1 -14848.763,E2 -14848.763} C_VEL
LIN {X 0,Y 325.363,Z 696.37,A -85,B 0,C 180,E1 -14850,E2 -14850} C_VEL
LIN {X 0,Y 325.318,Z 696.535,A -85,B 0,C 180,E1 -14851.238,E2 -14851.238} C_VEL
LIN {X 0,Y 325.217,Z 696.262,A -85,B 0,C 180,E1 -14852.478,E2 -14852.478} C_VEL
LIN {X 0,Y 325.079,Z 695.515,A -85,B 0,C 180,E1 -14853.719,E2 -14853.719} C_VEL
LIN {X 0,Y 324.991,Z 693.235,A -85,B 0,C 180,E1 -14855.866,E2 -14855.866} C_VEL
LIN {X 0,Y 325.216,Z 689.51,A -85,B 0,C 180,E1 -14858.075,E2 -14858.075} C_VEL
LIN {X 0,Y 325.569,Z 685.167,A -85,B 0,C 180,E1 -14859.945,E2 -14859.945} C_VEL
LIN {X 0,Y 326.35,Z 678.608,A -85,B 0,C 180,E1 -14862.121,E2 -14862.121} C_VEL
LIN {X 0,Y 327.401,Z 671.522,A -85,B 0,C 180,E1 -14863.975,E2 -14863.975} C_VEL
LIN {X 0,Y 328.782,Z 662.576,A -85,B 0,C 180,E1 -14865.863,E2 -14865.863} C_VEL
LIN {X 0,Y 330.366,Z 652.949,A -85,B 0,C 180,E1 -14867.487,E2 -14867.487} C_VEL
LIN {X 0,Y 332.316,Z 640.768,A -85,B 0,C 180,E1 -14869.136,E2 -14869.136} C_VEL
LIN {X 0,Y 334.256,Z 628.171,A -85,B 0,C 180,E1 -14870.461,E2 -14870.461} C_VEL
LIN {X 0,Y 335.969,Z 615.757,A -85,B 0,C 180,E1 -14871.474,E2 -14871.474} C_VEL
LIN {X 0,Y 337.54,Z 602.811,A -85,B 0,C 180,E1 -14872.253,E2 -14872.253} C_VEL
LIN {X 0,Y 338.621,Z 588.94,A -85,B 0,C 180,E1 -14872.862,E2 -14872.862} C_VEL
LIN {X 0,Y 341.539,Z 528.977,A -85,B 0,C 180,E1 -14874.639,E2 -14874.639} C_VEL
LIN {X 0,Y 340.213,Z 514.001,A -85,B 0,C 180,E1 -14875.34,E2 -14875.34} C_VEL
LIN {X 0,Y 338.123,Z 499.818,A -85,B 0,C 180,E1 -14876.124,E2 -14876.124} C_VEL
LIN {X 0,Y 335.014,Z 484.264,A -85,B 0,C 180,E1 -14877.154,E2 -14877.154} C_VEL
LIN {X 0,Y 333.582,Z 477.589,A -85,B 0,C 180,E1 -14877.652,E2 -14877.652} C_VEL
LIN {X 0,Y 334.214,Z 473.905,A -85,B 0,C 180,E1 -14878.581,E2 -14878.581} C_VEL
LIN {X 0,Y 333.056,Z 466.713,A -85,B 0,C 180,E1 -14880.779,E2 -14880.779} C_VEL
LIN {X 0,Y 330.833,Z 457.18,A -85,B 0,C 180,E1 -14884.056,E2 -14884.056} C_VEL
LIN {X 0,Y 328.947,Z 450.387,A -85,B 0,C 180,E1 -14886.744,E2 -14886.744} C_VEL
LIN {X 0,Y 326.609,Z 442.802,A -85,B 0,C 180,E1 -14890.321,E2 -14890.321} C_VEL
LIN {X 0,Y 326.581,Z 442.804,A -85,B 0,C 180,E1 -14893.523,E2 -14893.523} C_VEL
LIN {X 0,Y 326.584,Z 442.803,A -85,B 0,C 180,E1 -14897.027,E2 -14897.027} C_VEL
LIN {X 0,Y 326.615,Z 442.8,A -85,B 0,C 180,E1 -14900.773,E2 -14900.773} C_VEL
LIN {X 0,Y 326.617,Z 442.802,A -85,B 0,C 180,E1 -14904.481,E2 -14904.481} C_VEL
LIN {X 0,Y 326.611,Z 442.796,A -85,B 0,C 180,E1 -14907.456,E2 -14907.456} C_VEL
LIN {X 0,Y 326.62,Z 442.798,A -85,B 0,C 180,E1 -14910.337,E2 -14910.337} C_VEL
LIN {X 0,Y 326.605,Z 442.802,A -85,B 0,C 180,E1 -14914.509,E2 -14914.509} C_VEL
LIN {X 0,Y 326.605,Z 442.804,A -85,B 0,C 180,E1 -14918.542,E2 -14918.542} C_VEL
LIN {X 0,Y 326.621,Z 442.8,A -85,B 0,C 180,E1 -14922.468,E2 -14922.468} C_VEL
LIN {X 0,Y 326.692,Z 442.941,A -85,B 0,C 180,E1 -14924.88,E2 -14924.88} C_VEL
LIN {X 0,Y 327.596,Z 446.028,A -85,B 0,C 180,E1 -14926.561,E2 -14926.561} C_VEL
LIN {X 0,Y 329.975,Z 449.645,A -85,B 0,C 180,E1 -14927.108,E2 -14927.108} C_VEL
LIN {X 0,Y 335.75,Z 459.115,A -85,B 0,C 180,E1 -14928.392,E2 -14928.392} C_VEL
LIN {X 0,Y 341.665,Z 470.07,A -85,B 0,C 180,E1 -14929.645,E2 -14929.645} C_VEL
LIN {X 0,Y 343.696,Z 474.48,A -85,B 0,C 180,E1 -14930.064,E2 -14930.064} C_VEL
LIN {X 0,Y 339.744,Z 549.549,A -85,B 0,C 180,E1 -14932.347,E2 -14932.347} C_VEL
LIN {X 0,Y 338.832,Z 564.275,A -85,B 0,C 180,E1 -14933.075,E2 -14933.075} C_VEL
LIN {X 0,Y 337.682,Z 577.612,A -85,B 0,C 180,E1 -14934.027,E2 -14934.027} C_VEL
LIN {X 0,Y 336.313,Z 588.847,A -85,B 0,C 180,E1 -14935.055,E2 -14935.055} C_VEL
LIN {X 0,Y 334.924,Z 599.057,A -85,B 0,C 180,E1 -14936.24,E2 -14936.24} C_VEL
LIN {X 0,Y 333.43,Z 608.481,A -85,B 0,C 180,E1 -14937.584,E2 -14937.584} C_VEL
LIN {X 0,Y 331.985,Z 617.086,A -85,B 0,C 180,E1 -14939.09,E2 -14939.09} C_VEL
LIN {X 0,Y 330.551,Z 624.935,A -85,B 0,C 180,E1 -14940.76,E2 -14940.76} C_VEL
LIN {X 0,Y 329.346,Z 631.336,A -85,B 0,C 180,E1 -14942.446,E2 -14942.446} C_VEL
LIN {X 0,Y 328.186,Z 636.937,A -85,B 0,C 180,E1 -14944.298,E2 -14944.298} C_VEL
LIN {X 0,Y 327.259,Z 641.291,A -85,B 0,C 180,E1 -14946.164,E2 -14946.164} C_VEL
LIN {X 0,Y 326.543,Z 644.595,A -85,B 0,C 180,E1 -14948.093,E2 -14948.093} C_VEL
LIN {X 0,Y 325.958,Z 646.74,A -85,B 0,C 180,E1 -14949.932,E2 -14949.932} C_VEL
LIN {X 0,Y 325.683,Z 647.641,A -85,B 0,C 180,E1 -14951.199,E2 -14951.199} C_VEL
LIN {X 0,Y 325.496,Z 648.121,A -85,B 0,C 180,E1 -14952.469,E2 -14952.469} C_VEL
LIN {X 0,Y 325.353,Z 648.14,A -85,B 0,C 180,E1 -14953.746,E2 -14953.746} C_VEL
LIN {X 0,Y 325.23,Z 647.695,A -85,B 0,C 180,E1 -14955.029,E2 -14955.029} C_VEL
LIN {X 0,Y 325.197,Z 646.814,A -85,B 0,C 180,E1 -14956.317,E2 -14956.317} C_VEL
LIN {X 0,Y 325.295,Z 644.829,A -85,B 0,C 180,E1 -14958.079,E2 -14958.079} C_VEL
LIN {X 0,Y 325.505,Z 641.248,A -85,B 0,C 180,E1 -14960.21,E2 -14960.21} C_VEL
LIN {X 0,Y 325.848,Z 636.382,A -85,B 0,C 180,E1 -14962.267,E2 -14962.267} C_VEL
LIN {X 0,Y 326.314,Z 630.588,A -85,B 0,C 180,E1 -14964.155,E2 -14964.155} C_VEL
LIN {X 0,Y 326.998,Z 622.907,A -85,B 0,C 180,E1 -14966.142,E2 -14966.142} C_VEL
LIN {X 0,Y 327.713,Z 614.888,A -85,B 0,C 180,E1 -14967.804,E2 -14967.804} C_VEL
LIN {X 0,Y 328.611,Z 605.003,A -85,B 0,C 180,E1 -14969.466,E2 -14969.466} C_VEL
LIN {X 0,Y 329.48,Z 594.304,A -85,B 0,C 180,E1 -14970.923,E2 -14970.923} C_VEL
LIN {X 0,Y 330.397,Z 583.197,A -85,B 0,C 180,E1 -14972.126,E2 -14972.126} C_VEL
LIN {X 0,Y 331.184,Z 570.527,A -85,B 0,C 180,E1 -14973.214,E2 -14973.214} C_VEL
LIN {X 0,Y 331.936,Z 557.155,A -85,B 0,C 180,E1 -14974.059,E2 -14974.059} C_VEL
LIN {X 0,Y 332.379,Z 543.733,A -85,B 0,C 180,E1 -14974.654,E2 -14974.654} C_VEL
LIN {X 0,Y 334.567,Z 465.262,A -85,B 0,C 180,E1 -14976.787,E2 -14976.787} C_VEL
LIN {X 0,Y 326.62,Z 442.798,A -85,B 0,C 180,E1 -14977.871,E2 -14977.871} C_VEL
LIN {X 0,Y 326.564,Z 442.805,A -85,B 0,C 180,E1 -14981.848,E2 -14981.848} C_VEL
LIN {X 0,Y 326.528,Z 442.808,A -85,B 0,C 180,E1 -14985.257,E2 -14985.257} C_VEL
LIN {X 0,Y 326.564,Z 442.807,A -85,B 0,C 180,E1 -14988.152,E2 -14988.152} C_VEL
LIN {X 0,Y 326.569,Z 442.803,A -85,B 0,C 180,E1 -14991.383,E2 -14991.383} C_VEL
LIN {X 0,Y 326.621,Z 442.798,A -85,B 0,C 180,E1 -14994.851,E2 -14994.851} C_VEL
LIN {X 0,Y 326.61,Z 442.798,A -85,B 0,C 180,E1 -14997.455,E2 -14997.455} C_VEL
LIN {X 0,Y 326.619,Z 442.802,A -85,B 0,C 180,E1 -15000.336,E2 -15000.336} C_VEL
LIN {X 0,Y 326.643,Z 442.797,A -85,B 0,C 180,E1 -15004.644,E2 -15004.644} C_VEL
LIN {X 0,Y 326.64,Z 442.799,A -85,B 0,C 180,E1 -15008.544,E2 -15008.544} C_VEL
LIN {X 0,Y 326.746,Z 442.781,A -85,B 0,C 180,E1 -15011.177,E2 -15011.177} C_VEL
LIN {X 0,Y 326.765,Z 442.778,A -85,B 0,C 180,E1 -15015.433,E2 -15015.433} C_VEL
LIN {X 0,Y 326.76,Z 442.781,A -85,B 0,C 180,E1 -15018.838,E2 -15018.838} C_VEL
LIN {X 0,Y 326.915,Z 442.764,A -85,B 0,C 180,E1 -15022.588,E2 -15022.588} C_VEL
LIN {X 0,Y 326.762,Z 442.78,A -85,B 0,C 180,E1 -15025.064,E2 -15025.064} C_VEL
LIN {X 0,Y 327.043,Z 442.744,A -85,B 0,C 180,E1 -15027.536,E2 -15027.536} C_VEL
LIN {X 0,Y 327.142,Z 442.733,A -85,B 0,C 180,E1 -15030,E2 -15030} C_VEL
LIN {X 0,Y 327.034,Z 442.751,A -85,B 0,C 180,E1 -15032.463,E2 -15032.463} C_VEL
LIN {X 0,Y 326.983,Z 442.754,A -85,B 0,C 180,E1 -15036.169,E2 -15036.169} C_VEL
LIN {X 0,Y 326.805,Z 442.774,A -85,B 0,C 180,E1 -15039.906,E2 -15039.906} C_VEL
LIN {X 0,Y 326.76,Z 442.779,A -85,B 0,C 180,E1 -15043.685,E2 -15043.685} C_VEL
LIN {X 0,Y 326.664,Z 442.791,A -85,B 0,C 180,E1 -15047.529,E2 -15047.529} C_VEL
LIN {X 0,Y 326.631,Z 442.797,A -85,B 0,C 180,E1 -15050.137,E2 -15050.137} C_VEL
LIN {X 0,Y 326.639,Z 442.796,A -85,B 0,C 180,E1 -15054.129,E2 -15054.129} C_VEL
LIN {X 0,Y 326.621,Z 442.799,A -85,B 0,C 180,E1 -15058.253,E2 -15058.253} C_VEL
LIN {X 0,Y 326.573,Z 442.804,A -85,B 0,C 180,E1 -15061.097,E2 -15061.097} C_VEL
LIN {X 0,Y 326.606,Z 442.799,A -85,B 0,C 180,E1 -15064.019,E2 -15064.019} C_VEL
LIN {X 0,Y 326.622,Z 442.797,A -85,B 0,C 180,E1 -15067.237,E2 -15067.237} C_VEL
LIN {X 0,Y 326.543,Z 442.807,A -85,B 0,C 180,E1 -15071.124,E2 -15071.124} C_VEL
LIN {X 0,Y 326.56,Z 442.804,A -85,B 0,C 180,E1 -15073.525,E2 -15073.525} C_VEL
LIN {X 0,Y 326.574,Z 442.804,A -85,B 0,C 180,E1 -15077.028,E2 -15077.028} C_VEL
LIN {X 0,Y 326.609,Z 442.802,A -85,B 0,C 180,E1 -15080.773,E2 -15080.773} C_VEL
LIN {X 0,Y 326.612,Z 442.802,A -85,B 0,C 180,E1 -15084.48,E2 -15084.48} C_VEL
LIN {X 0,Y 326.604,Z 442.799,A -85,B 0,C 180,E1 -15086.83,E2 -15086.83} C_VEL
LIN {X 0,Y 325.971,Z 442.88,A -85,B 0,C 180,E1 -15087.859,E2 -15087.859} C_VEL
LIN {X 0,Y 323.126,Z 443.232,A -85,B 0,C 180,E1 -15089.533,E2 -15089.533} C_VEL
LIN {X 0,Y 320.702,Z 443.537,A -85,B 0,C 180,E1 -15090.889,E2 -15090.889} C_VEL
LIN {X 0,Y 319.675,Z 443.663,A -85,B 0,C 180,E1 -15091.939,E2 -15091.939} C_VEL
LIN {X 0,Y 319.599,Z 443.674,A -85,B 0,C 180,E1 -15092.295,E2 -15092.295} C_VEL
LIN {X 0,Y 319.604,Z 443.671,A -85,B 0,C 180,E1 -15095.304,E2 -15095.304} C_VEL
LIN {X 0,Y 319.597,Z 443.672,A -85,B 0,C 180,E1 -15098.048,E2 -15098.048} C_VEL
LIN {X 0,Y 319.688,Z 443.663,A -85,B 0,C 180,E1 -15100.962,E2 -15100.962} C_VEL
LIN {X 0,Y 319.73,Z 443.655,A -85,B 0,C 180,E1 -15105.276,E2 -15105.276} C_VEL
LIN {X 0,Y 319.755,Z 443.652,A -85,B 0,C 180,E1 -15109.873,E2 -15109.873} C_VEL
LIN {X 0,Y 319.92,Z 443.635,A -85,B 0,C 180,E1 -15112.426,E2 -15112.426} C_VEL
LIN {X 0,Y 319.74,Z 443.656,A -85,B 0,C 180,E1 -15114.956,E2 -15114.956} C_VEL
LIN {X 0,Y 319.988,Z 443.623,A -85,B 0,C 180,E1 -15117.482,E2 -15117.482} C_VEL
LIN {X 0,Y 320.148,Z 443.603,A -85,B 0,C 180,E1 -15120,E2 -15120} C_VEL
LIN {X 0,Y 319.99,Z 443.627,A -85,B 0,C 180,E1 -15122.518,E2 -15122.518} C_VEL
LIN {X 0,Y 319.951,Z 443.63,A -85,B 0,C 180,E1 -15126.306,E2 -15126.306} C_VEL
LIN {X 0,Y 319.842,Z 443.645,A -85,B 0,C 180,E1 -15128.848,E2 -15128.848} C_VEL
LIN {X 0,Y 319.682,Z 443.666,A -85,B 0,C 180,E1 -15132.7,E2 -15132.7} C_VEL
LIN {X 0,Y 319.699,Z 443.659,A -85,B 0,C 180,E1 -15135.296,E2 -15135.296} C_VEL
LIN {X 0,Y 319.673,Z 443.663,A -85,B 0,C 180,E1 -15139.255,E2 -15139.255} C_VEL
LIN {X 0,Y 319.559,Z 443.677,A -85,B 0,C 180,E1 -15143.32,E2 -15143.32} C_VEL
LIN {X 0,Y 319.634,Z 443.668,A -85,B 0,C 180,E1 -15146.088,E2 -15146.088} C_VEL
LIN {X 0,Y 319.589,Z 443.676,A -85,B 0,C 180,E1 -15148.934,E2 -15148.934} C_VEL
LIN {X 0,Y 319.532,Z 443.679,A -85,B 0,C 180,E1 -15151.862,E2 -15151.862} C_VEL
LIN {X 0,Y 319.579,Z 443.674,A -85,B 0,C 180,E1 -15155.543,E2 -15155.543} C_VEL
LIN {X 0,Y 319.557,Z 443.677,A -85,B 0,C 180,E1 -15158.011,E2 -15158.011} C_VEL
LIN {X 0,Y 319.525,Z 443.68,A -85,B 0,C 180,E1 -15161.597,E2 -15161.597} C_VEL
LIN {X 0,Y 319.516,Z 443.687,A -85,B 0,C 180,E1 -15164.738,E2 -15164.738} C_VEL
LIN {X 0,Y 319.526,Z 443.683,A -85,B 0,C 180,E1 -15168.403,E2 -15168.403} C_VEL
LIN {X 0,Y 319.543,Z 443.678,A -85,B 0,C 180,E1 -15171.988,E2 -15171.988} C_VEL
LIN {X 0,Y 319.564,Z 443.68,A -85,B 0,C 180,E1 -15175.124,E2 -15175.124} C_VEL
LIN {X 0,Y 319.613,Z 443.775,A -85,B 0,C 180,E1 -15176.677,E2 -15176.677} C_VEL
LIN {X 0,Y 322.78,Z 458.839,A -85,B 0,C 180,E1 -15180.568,E2 -15180.568} C_VEL
LIN {X 0,Y 324.276,Z 466.795,A -85,B 0,C 180,E1 -15182.548,E2 -15182.548} C_VEL
LIN {X 0,Y 322.24,Z 484.561,A -85,B 0,C 180,E1 -15186.62,E2 -15186.62} C_VEL
LIN {X 0,Y 326.894,Z 529.185,A -85,B 0,C 180,E1 -15188.202,E2 -15188.202} C_VEL
LIN {X 0,Y 325.054,Z 594.487,A -85,B 0,C 180,E1 -15190.05,E2 -15190.05} C_VEL
LIN {X 0,Y 324.279,Z 607.778,A -85,B 0,C 180,E1 -15190.66,E2 -15190.66} C_VEL
LIN {X 0,Y 323.432,Z 620.184,A -85,B 0,C 180,E1 -15191.471,E2 -15191.471} C_VEL
LIN {X 0,Y 322.496,Z 631.004,A -85,B 0,C 180,E1 -15192.4,E2 -15192.4} C_VEL
LIN {X 0,Y 321.468,Z 642.515,A -85,B 0,C 180,E1 -15193.652,E2 -15193.652} C_VEL
LIN {X 0,Y 320.422,Z 652.981,A -85,B 0,C 180,E1 -15195.069,E2 -15195.069} C_VEL
LIN {X 0,Y 319.772,Z 660.653,A -85,B 0,C 180,E1 -15196.334,E2 -15196.334} C_VEL
LIN {X 0,Y 319.121,Z 668.73,A -85,B 0,C 180,E1 -15197.924,E2 -15197.924} C_VEL
LIN {X 0,Y 318.535,Z 676.56,A -85,B 0,C 180,E1 -15199.834,E2 -15199.834} C_VEL
LIN {X 0,Y 318.244,Z 682.824,A -85,B 0,C 180,E1 -15201.747,E2 -15201.747} C_VEL
LIN {X 0,Y 318.172,Z 687.867,A -85,B 0,C 180,E1 -15203.718,E2 -15203.718} C_VEL
LIN {X 0,Y 318.139,Z 691.402,A -85,B 0,C 180,E1 -15205.566,E2 -15205.566} C_VEL
LIN {X 0,Y 318.294,Z 693.968,A -85,B 0,C 180,E1 -15207.469,E2 -15207.469} C_VEL
LIN {X 0,Y 318.294,Z 695.098,A -85,B 0,C 180,E1 -15208.735,E2 -15208.735} C_VEL
LIN {X 0,Y 318.299,Z 695.738,A -85,B 0,C 180,E1 -15210,E2 -15210} C_VEL
LIN {X 0,Y 318.254,Z 695.945,A -85,B 0,C 180,E1 -15211.266,E2 -15211.266} C_VEL
LIN {X 0,Y 318.122,Z 695.717,A -85,B 0,C 180,E1 -15212.533,E2 -15212.533} C_VEL
LIN {X 0,Y 317.998,Z 695.042,A -85,B 0,C 180,E1 -15213.802,E2 -15213.802} C_VEL
LIN {X 0,Y 317.905,Z 693.057,A -85,B 0,C 180,E1 -15215.829,E2 -15215.829} C_VEL
LIN {X 0,Y 318.16,Z 689.193,A -85,B 0,C 180,E1 -15218.256,E2 -15218.256} C_VEL
LIN {X 0,Y 318.534,Z 684.961,A -85,B 0,C 180,E1 -15220.167,E2 -15220.167} C_VEL
LIN {X 0,Y 319.22,Z 679.563,A -85,B 0,C 180,E1 -15222.073,E2 -15222.073} C_VEL
LIN {X 0,Y 320.315,Z 672.852,A -85,B 0,C 180,E1 -15223.967,E2 -15223.967} C_VEL
LIN {X 0,Y 321.572,Z 665.106,A -85,B 0,C 180,E1 -15225.737,E2 -15225.737} C_VEL
LIN {X 0,Y 323.106,Z 656.211,A -85,B 0,C 180,E1 -15227.403,E2 -15227.403} C_VEL
LIN {X 0,Y 324.9,Z 646.169,A -85,B 0,C 180,E1 -15228.934,E2 -15228.934} C_VEL
LIN {X 0,Y 326.794,Z 635.137,A -85,B 0,C 180,E1 -15230.291,E2 -15230.291} C_VEL
LIN {X 0,Y 328.647,Z 622.855,A -85,B 0,C 180,E1 -15231.483,E2 -15231.483} C_VEL
LIN {X 0,Y 330.425,Z 610.126,A -85,B 0,C 180,E1 -15232.429,E2 -15232.429} C_VEL
LIN {X 0,Y 331.971,Z 596.263,A -85,B 0,C 180,E1 -15233.182,E2 -15233.182} C_VEL
LIN {X 0,Y 332.888,Z 583.127,A -85,B 0,C 180,E1 -15233.684,E2 -15233.684} C_VEL
LIN {X 0,Y 335.658,Z 530.057,A -85,B 0,C 180,E1 -15235.289,E2 -15235.289} C_VEL
LIN {X 0,Y 334.519,Z 516.302,A -85,B 0,C 180,E1 -15235.951,E2 -15235.951} C_VEL
LIN {X 0,Y 332.59,Z 502.158,A -85,B 0,C 180,E1 -15236.769,E2 -15236.769} C_VEL
LIN {X 0,Y 329.642,Z 486.981,A -85,B 0,C 180,E1 -15237.8,E2 -15237.8} C_VEL
LIN {X 0,Y 327.451,Z 476.689,A -85,B 0,C 180,E1 -15238.619,E2 -15238.619} C_VEL
LIN {X 0,Y 327.037,Z 472.265,A -85,B 0,C 180,E1 -15239.952,E2 -15239.952} C_VEL
LIN {X 0,Y 325.359,Z 464.138,A -85,B 0,C 180,E1 -15242.686,E2 -15242.686} C_VEL
LIN {X 0,Y 323.494,Z 456.623,A -85,B 0,C 180,E1 -15245.532,E2 -15245.532} C_VEL
LIN {X 0,Y 321.701,Z 450.69,A -85,B 0,C 180,E1 -15248.143,E2 -15248.143} C_VEL
LIN {X 0,Y 320.142,Z 445.678,A -85,B 0,C 180,E1 -15250.662,E2 -15250.662} C_VEL
LIN {X 0,Y 319.535,Z 443.683,A -85,B 0,C 180,E1 -15251.864,E2 -15251.864} C_VEL
LIN {X 0,Y 319.518,Z 443.683,A -85,B 0,C 180,E1 -15255.262,E2 -15255.262} C_VEL
LIN {X 0,Y 319.532,Z 443.683,A -85,B 0,C 180,E1 -15258.712,E2 -15258.712} C_VEL
LIN {X 0,Y 319.581,Z 443.679,A -85,B 0,C 180,E1 -15262.344,E2 -15262.344} C_VEL
LIN {X 0,Y 319.564,Z 443.675,A -85,B 0,C 180,E1 -15265.124,E2 -15265.124} C_VEL
LIN {X 0,Y 319.528,Z 443.68,A -85,B 0,C 180,E1 -15268.138,E2 -15268.138} C_VEL
LIN {X 0,Y 319.574,Z 443.674,A -85,B 0,C 180,E1 -15271.604,E2 -15271.604} C_VEL
LIN {X 0,Y 319.531,Z 443.682,A -85,B 0,C 180,E1 -15275.298,E2 -15275.298} C_VEL
LIN {X 0,Y 319.563,Z 443.678,A -85,B 0,C 180,E1 -15278.045,E2 -15278.045} C_VEL
LIN {X 0,Y 319.574,Z 443.68,A -85,B 0,C 180,E1 -15282.068,E2 -15282.068} C_VEL
LIN {X 0,Y 319.586,Z 443.825,A -85,B 0,C 180,E1 -15283.388,E2 -15283.388} C_VEL
LIN {X 0,Y 320.584,Z 447.041,A -85,B 0,C 180,E1 -15285.361,E2 -15285.361} C_VEL
LIN {X 0,Y 322.856,Z 450.504,A -85,B 0,C 180,E1 -15285.946,E2 -15285.946} C_VEL
LIN {X 0,Y 328.489,Z 459.048,A -85,B 0,C 180,E1 -15287.284,E2 -15287.284} C_VEL
LIN {X 0,Y 334.65,Z 470.045,A -85,B 0,C 180,E1 -15288.685,E2 -15288.685} C_VEL
LIN {X 0,Y 337.957,Z 476.844,A -85,B 0,C 180,E1 -15289.414,E2 -15289.414} C_VEL
LIN {X 0,Y 333.78,Z 550.513,A -85,B 0,C 180,E1 -15291.714,E2 -15291.714} C_VEL
LIN {X 0,Y 332.871,Z 564.396,A -85,B 0,C 180,E1 -15292.417,E2 -15292.417} C_VEL
LIN {X 0,Y 331.706,Z 576.9,A -85,B 0,C 180,E1 -15293.308,E2 -15293.308} C_VEL
LIN {X 0,Y 330.072,Z 589.737,A -85,B 0,C 180,E1 -15294.502,E2 -15294.502} C_VEL
LIN {X 0,Y 328.414,Z 601.019,A -85,B 0,C 180,E1 -15295.858,E2 -15295.858} C_VEL
LIN {X 0,Y 326.853,Z 610.246,A -85,B 0,C 180,E1 -15297.227,E2 -15297.227} C_VEL
LIN {X 0,Y 325.346,Z 618.682,A -85,B 0,C 180,E1 -15298.762,E2 -15298.762} C_VEL
LIN {X 0,Y 323.745,Z 626.702,A -85,B 0,C 180,E1 -15300.566,E2 -15300.566} C_VEL
LIN {X 0,Y 322.3,Z 633.512,A -85,B 0,C 180,E1 -15302.499,E2 -15302.499} C_VEL
LIN {X 0,Y 321.107,Z 638.798,A -85,B 0,C 180,E1 -15304.393,E2 -15304.393} C_VEL
LIN {X 0,Y 320.171,Z 642.862,A -85,B 0,C 180,E1 -15306.301,E2 -15306.301} C_VEL
LIN {X 0,Y 319.484,Z 645.713,A -85,B 0,C 180,E1 -15308.142,E2 -15308.142} C_VEL
LIN {X 0,Y 318.853,Z 647.753,A -85,B 0,C 180,E1 -15310.156,E2 -15310.156} C_VEL
LIN {X 0,Y 318.569,Z 648.5,A -85,B 0,C 180,E1 -15311.452,E2 -15311.452} C_VEL
LIN {X 0,Y 318.281,Z 648.695,A -85,B 0,C 180,E1 -15313.693,E2 -15313.693} C_VEL
LIN {X 0,Y 318.135,Z 648.012,A -85,B 0,C 180,E1 -15315.373,E2 -15315.373} C_VEL
LIN {X 0,Y 318.128,Z 646.912,A -85,B 0,C 180,E1 -15316.69,E2 -15316.69} C_VEL
LIN {X 0,Y 318.224,Z 645.037,A -85,B 0,C 180,E1 -15318.256,E2 -15318.256} C_VEL
LIN {X 0,Y 318.387,Z 642.087,A -85,B 0,C 180,E1 -15320.007,E2 -15320.007} C_VEL
LIN {X 0,Y 318.75,Z 637.161,A -85,B 0,C 180,E1 -15322.173,E2 -15322.173} C_VEL
LIN {X 0,Y 319.275,Z 630.479,A -85,B 0,C 180,E1 -15324.377,E2 -15324.377} C_VEL
LIN {X 0,Y 320.018,Z 622.587,A -85,B 0,C 180,E1 -15326.405,E2 -15326.405} C_VEL
LIN {X 0,Y 320.753,Z 614.35,A -85,B 0,C 180,E1 -15328.105,E2 -15328.105} C_VEL
LIN {X 0,Y 321.715,Z 604.426,A -85,B 0,C 180,E1 -15329.773,E2 -15329.773} C_VEL
LIN {X 0,Y 322.519,Z 594.199,A -85,B 0,C 180,E1 -15331.167,E2 -15331.167} C_VEL
LIN {X 0,Y 323.525,Z 582.049,A -85,B 0,C 180,E1 -15332.487,E2 -15332.487} C_VEL
LIN {X 0,Y 324.348,Z 569.595,A -85,B 0,C 180,E1 -15333.541,E2 -15333.541} C_VEL
LIN {X 0,Y 325.097,Z 555.368,A -85,B 0,C 180,E1 -15334.426,E2 -15334.426} C_VEL
LIN {X 0,Y 325.533,Z 542.138,A -85,B 0,C 180,E1 -15334.982,E2 -15334.982} C_VEL
LIN {X 0,Y 327.699,Z 466.749,A -85,B 0,C 180,E1 -15337.086,E2 -15337.086} C_VEL
LIN {X 0,Y 319.582,Z 443.678,A -85,B 0,C 180,E1 -15338.22,E2 -15338.22} C_VEL
LIN {X 0,Y 319.554,Z 443.678,A -85,B 0,C 180,E1 -15342.983,E2 -15342.983} C_VEL
LIN {X 0,Y 319.554,Z 443.678,A -85,B 0,C 180,E1 -15347.016,E2 -15347.016} C_VEL
LIN {X 0,Y 319.547,Z 443.683,A -85,B 0,C 180,E1 -15350.37,E2 -15350.37} C_VEL
LIN {X 0,Y 319.582,Z 443.679,A -85,B 0,C 180,E1 -15354.457,E2 -15354.457} C_VEL
LIN {X 0,Y 319.526,Z 443.683,A -85,B 0,C 180,E1 -15358.137,E2 -15358.137} C_VEL
LIN {X 0,Y 319.573,Z 443.674,A -85,B 0,C 180,E1 -15361.603,E2 -15361.603} C_VEL
LIN {X 0,Y 319.576,Z 443.674,A -85,B 0,C 180,E1 -15365.301,E2 -15365.301} C_VEL
LIN {X 0,Y 319.593,Z 443.674,A -85,B 0,C 180,E1 -15368.047,E2 -15368.047} C_VEL
LIN {X 0,Y 319.691,Z 443.661,A -85,B 0,C 180,E1 -15370.962,E2 -15370.962} C_VEL
LIN {X 0,Y 319.733,Z 443.655,A -85,B 0,C 180,E1 -15375.275,E2 -15375.275} C_VEL
LIN {X 0,Y 319.717,Z 443.661,A -85,B 0,C 180,E1 -15378.589,E2 -15378.589} C_VEL
LIN {X 0,Y 319.855,Z 443.645,A -85,B 0,C 180,E1 -15382.424,E2 -15382.424} C_VEL
LIN {X 0,Y 319.73,Z 443.656,A -85,B 0,C 180,E1 -15384.955,E2 -15384.955} C_VEL
LIN {X 0,Y 319.986,Z 443.623,A -85,B 0,C 180,E1 -15387.482,E2 -15387.482} C_VEL
LIN {X 0,Y 320.096,Z 443.611,A -85,B 0,C 180,E1 -15390,E2 -15390} C_VEL
LIN {X 0,Y 319.978,Z 443.63,A -85,B 0,C 180,E1 -15392.517,E2 -15392.517} C_VEL
LIN {X 0,Y 319.937,Z 443.633,A -85,B 0,C 180,E1 -15396.305,E2 -15396.305} C_VEL
LIN {X 0,Y 319.752,Z 443.654,A -85,B 0,C 180,E1 -15400.127,E2 -15400.127} C_VEL
LIN {X 0,Y 319.733,Z 443.656,A -85,B 0,C 180,E1 -15403.992,E2 -15403.992} C_VEL
LIN {X 0,Y 319.624,Z 443.669,A -85,B 0,C 180,E1 -15407.928,E2 -15407.928} C_VEL
LIN {X 0,Y 319.568,Z 443.676,A -85,B 0,C 180,E1 -15411.954,E2 -15411.954} C_VEL
LIN {X 0,Y 319.573,Z 443.676,A -85,B 0,C 180,E1 -15416.093,E2 -15416.093} C_VEL
LIN {X 0,Y 319.552,Z 443.679,A -85,B 0,C 180,E1 -15418.937,E2 -15418.937} C_VEL
LIN {X 0,Y 319.523,Z 443.681,A -85,B 0,C 180,E1 -15421.862,E2 -15421.862} C_VEL
LIN {X 0,Y 319.578,Z 443.674,A -85,B 0,C 180,E1 -15425.542,E2 -15425.542} C_VEL
LIN {X 0,Y 319.526,Z 443.68,A -85,B 0,C 180,E1 -15429.662,E2 -15429.662} C_VEL
LIN {X 0,Y 319.519,Z 443.681,A -85,B 0,C 180,E1 -15433.46,E2 -15433.46} C_VEL
LIN {X 0,Y 319.552,Z 443.679,A -85,B 0,C 180,E1 -15437.016,E2 -15437.016} C_VEL
LIN {X 0,Y 319.545,Z 443.682,A -85,B 0,C 180,E1 -15440.371,E2 -15440.371} C_VEL
LIN {X 0,Y 319.579,Z 443.678,A -85,B 0,C 180,E1 -15444.457,E2 -15444.457} C_VEL
LIN {X 0,Y 319.529,Z 443.681,A -85,B 0,C 180,E1 -15448.138,E2 -15448.138} C_VEL
LIN {X 0,Y 319.61,Z 443.67,A -85,B 0,C 180,E1 -15451.59,E2 -15451.59} C_VEL
LIN {X 0,Y 319.599,Z 443.674,A -85,B 0,C 180,E1 -15452.295,E2 -15452.295} C_VEL
LIN {X 0,Y 318.961,Z 443.759,A -85,B 0,C 180,E1 -15453.346,E2 -15453.346} C_VEL
LIN {X 0,Y 316.143,Z 444.111,A -85,B 0,C 180,E1 -15455.058,E2 -15455.058} C_VEL
LIN {X 0,Y 313.724,Z 444.407,A -85,B 0,C 180,E1 -15456.445,E2 -15456.445} C_VEL
LIN {X 0,Y 312.66,Z 444.535,A -85,B 0,C 180,E1 -15457.519,E2 -15457.519} C_VEL
LIN {X 0,Y 312.561,Z 444.546,A -85,B 0,C 180,E1 -15457.883,E2 -15457.883} C_VEL
LIN {X 0,Y 312.637,Z 444.538,A -85,B 0,C 180,E1 -15461.656,E2 -15461.656} C_VEL
LIN {X 0,Y 312.693,Z 444.531,A -85,B 0,C 180,E1 -15465.686,E2 -15465.686} C_VEL
LIN {X 0,Y 312.7,Z 444.53,A -85,B 0,C 180,E1 -15469.642,E2 -15469.642} C_VEL
LIN {X 0,Y 312.861,Z 444.513,A -85,B 0,C 180,E1 -15472.254,E2 -15472.254} C_VEL
LIN {X 0,Y 312.71,Z 444.533,A -85,B 0,C 180,E1 -15474.842,E2 -15474.842} C_VEL
LIN {X 0,Y 312.988,Z 444.5,A -85,B 0,C 180,E1 -15478.713,E2 -15478.713} C_VEL
LIN {X 0,Y 312.988,Z 444.495,A -85,B 0,C 180,E1 -15481.287,E2 -15481.287} C_VEL
LIN {X 0,Y 312.716,Z 444.53,A -85,B 0,C 180,E1 -15485.158,E2 -15485.158} C_VEL
LIN {X 0,Y 312.871,Z 444.509,A -85,B 0,C 180,E1 -15487.746,E2 -15487.746} C_VEL
LIN {X 0,Y 312.669,Z 444.534,A -85,B 0,C 180,E1 -15491.671,E2 -15491.671} C_VEL
LIN {X 0,Y 312.699,Z 444.534,A -85,B 0,C 180,E1 -15494.888,E2 -15494.888} C_VEL
LIN {X 0,Y 312.629,Z 444.541,A -85,B 0,C 180,E1 -15499.236,E2 -15499.236} C_VEL
LIN {X 0,Y 312.525,Z 444.557,A -85,B 0,C 180,E1 -15502.781,E2 -15502.781} C_VEL
LIN {X 0,Y 312.582,Z 444.551,A -85,B 0,C 180,E1 -15506.723,E2 -15506.723} C_VEL
LIN {X 0,Y 312.545,Z 444.55,A -85,B 0,C 180,E1 -15509.65,E2 -15509.65} C_VEL
LIN {X 0,Y 312.519,Z 444.553,A -85,B 0,C 180,E1 -15513.689,E2 -15513.689} C_VEL
LIN {X 0,Y 312.525,Z 444.553,A -85,B 0,C 180,E1 -15517.385,E2 -15517.385} C_VEL
LIN {X 0,Y 312.489,Z 444.562,A -85,B 0,C 180,E1 -15520.709,E2 -15520.709} C_VEL
LIN {X 0,Y 312.473,Z 444.56,A -85,B 0,C 180,E1 -15524.206,E2 -15524.206} C_VEL
LIN {X 0,Y 312.486,Z 444.557,A -85,B 0,C 180,E1 -15527.919,E2 -15527.919} C_VEL
LIN {X 0,Y 312.499,Z 444.559,A -85,B 0,C 180,E1 -15530.972,E2 -15530.972} C_VEL
LIN {X 0,Y 312.532,Z 444.553,A -85,B 0,C 180,E1 -15534.221,E2 -15534.221} C_VEL
LIN {X 0,Y 312.524,Z 444.595,A -85,B 0,C 180,E1 -15536.381,E2 -15536.381} C_VEL
LIN {X 0,Y 315.216,Z 457.408,A -85,B 0,C 180,E1 -15539.776,E2 -15539.776} C_VEL
LIN {X 0,Y 317.261,Z 467.591,A -85,B 0,C 180,E1 -15542.386,E2 -15542.386} C_VEL
LIN {X 0,Y 315.319,Z 484.139,A -85,B 0,C 180,E1 -15546.26,E2 -15546.26} C_VEL
LIN {X 0,Y 320.009,Z 529.862,A -85,B 0,C 180,E1 -15547.908,E2 -15547.908} C_VEL
LIN {X 0,Y 318.103,Z 594.452,A -85,B 0,C 180,E1 -15549.806,E2 -15549.806} C_VEL
LIN {X 0,Y 317.329,Z 607.542,A -85,B 0,C 180,E1 -15550.429,E2 -15550.429} C_VEL
LIN {X 0,Y 316.474,Z 619.309,A -85,B 0,C 180,E1 -15551.216,E2 -15551.216} C_VEL
LIN {X 0,Y 315.518,Z 630.185,A -85,B 0,C 180,E1 -15552.166,E2 -15552.166} C_VEL
LIN {X 0,Y 314.468,Z 641.732,A -85,B 0,C 180,E1 -15553.445,E2 -15553.445} C_VEL
LIN {X 0,Y 313.4,Z 652.401,A -85,B 0,C 180,E1 -15554.918,E2 -15554.918} C_VEL
LIN {X 0,Y 312.655,Z 660.834,A -85,B 0,C 180,E1 -15556.348,E2 -15556.348} C_VEL
LIN {X 0,Y 311.892,Z 670.161,A -85,B 0,C 180,E1 -15558.3,E2 -15558.3} C_VEL
LIN {X 0,Y 311.372,Z 677.648,A -85,B 0,C 180,E1 -15560.254,E2 -15560.254} C_VEL
LIN {X 0,Y 311.147,Z 683.573,A -85,B 0,C 180,E1 -15562.212,E2 -15562.212} C_VEL
LIN {X 0,Y 311.099,Z 688.194,A -85,B 0,C 180,E1 -15564.182,E2 -15564.182} C_VEL
LIN {X 0,Y 311.058,Z 691.549,A -85,B 0,C 180,E1 -15566.114,E2 -15566.114} C_VEL
LIN {X 0,Y 311.233,Z 693.202,A -85,B 0,C 180,E1 -15567.412,E2 -15567.412} C_VEL
LIN {X 0,Y 311.234,Z 694.39,A -85,B 0,C 180,E1 -15568.707,E2 -15568.707} C_VEL
LIN {X 0,Y 311.236,Z 695.107,A -85,B 0,C 180,E1 -15570,E2 -15570} C_VEL
LIN {X 0,Y 311.191,Z 695.354,A -85,B 0,C 180,E1 -15571.295,E2 -15571.295} C_VEL
LIN {X 0,Y 311.029,Z 695.164,A -85,B 0,C 180,E1 -15572.591,E2 -15572.591} C_VEL
LIN {X 0,Y 310.918,Z 694.557,A -85,B 0,C 180,E1 -15573.889,E2 -15573.889} C_VEL
LIN {X 0,Y 310.828,Z 692.834,A -85,B 0,C 180,E1 -15575.807,E2 -15575.807} C_VEL
LIN {X 0,Y 311.093,Z 688.913,A -85,B 0,C 180,E1 -15578.445,E2 -15578.445} C_VEL
LIN {X 0,Y 311.515,Z 684.769,A -85,B 0,C 180,E1 -15580.399,E2 -15580.399} C_VEL
LIN {X 0,Y 312.251,Z 679.462,A -85,B 0,C 180,E1 -15582.347,E2 -15582.347} C_VEL
LIN {X 0,Y 313.398,Z 672.896,A -85,B 0,C 180,E1 -15584.281,E2 -15584.281} C_VEL
LIN {X 0,Y 314.649,Z 665.845,A -85,B 0,C 180,E1 -15585.98,E2 -15585.98} C_VEL
LIN {X 0,Y 316.369,Z 656.677,A -85,B 0,C 180,E1 -15587.786,E2 -15587.786} C_VEL
LIN {X 0,Y 318.462,Z 645.721,A -85,B 0,C 180,E1 -15589.499,E2 -15589.499} C_VEL
LIN {X 0,Y 320.657,Z 633.394,A -85,B 0,C 180,E1 -15591.033,E2 -15591.033} C_VEL
LIN {X 0,Y 322.688,Z 620.998,A -85,B 0,C 180,E1 -15592.236,E2 -15592.236} C_VEL
LIN {X 0,Y 324.468,Z 609.163,A -85,B 0,C 180,E1 -15593.116,E2 -15593.116} C_VEL
LIN {X 0,Y 326.151,Z 594.458,A -85,B 0,C 180,E1 -15593.915,E2 -15593.915} C_VEL
LIN {X 0,Y 327.003,Z 581.914,A -85,B 0,C 180,E1 -15594.395,E2 -15594.395} C_VEL
LIN {X 0,Y 329.901,Z 531.569,A -85,B 0,C 180,E1 -15595.953,E2 -15595.953} C_VEL
LIN {X 0,Y 328.963,Z 518.763,A -85,B 0,C 180,E1 -15596.592,E2 -15596.592} C_VEL
LIN {X 0,Y 327.042,Z 504.175,A -85,B 0,C 180,E1 -15597.457,E2 -15597.457} C_VEL
LIN {X 0,Y 324.312,Z 489.344,A -85,B 0,C 180,E1 -15598.518,E2 -15598.518} C_VEL
LIN {X 0,Y 322.014,Z 479.472,A -85,B 0,C 180,E1 -15599.327,E2 -15599.327} C_VEL
LIN {X 0,Y 320.63,Z 475.751,A -85,B 0,C 180,E1 -15599.774,E2 -15599.774} C_VEL
LIN {X 0,Y 318.951,Z 467.189,A -85,B 0,C 180,E1 -15602.714,E2 -15602.714} C_VEL
LIN {X 0,Y 317.189,Z 459.87,A -85,B 0,C 180,E1 -15605.566,E2 -15605.566} C_VEL
LIN {X 0,Y 315.741,Z 454.989,A -85,B 0,C 180,E1 -15607.742,E2 -15607.742} C_VEL
LIN {X 0,Y 314.113,Z 449.603,A -85,B 0,C 180,E1 -15610.472,E2 -15610.472} C_VEL
LIN {X 0,Y 312.513,Z 444.556,A -85,B 0,C 180,E1 -15613.55,E2 -15613.55} C_VEL
LIN {X 0,Y 312.518,Z 444.555,A -85,B 0,C 180,E1 -15617.913,E2 -15617.913} C_VEL
LIN {X 0,Y 312.539,Z 444.553,A -85,B 0,C 180,E1 -15621.911,E2 -15621.911} C_VEL
LIN {X 0,Y 312.51,Z 444.553,A -85,B 0,C 180,E1 -15625.79,E2 -15625.79} C_VEL
LIN {X 0,Y 312.51,Z 444.557,A -85,B 0,C 180,E1 -15628.852,E2 -15628.852} C_VEL
LIN {X 0,Y 312.531,Z 444.551,A -85,B 0,C 180,E1 -15631.82,E2 -15631.82} C_VEL
LIN {X 0,Y 312.521,Z 444.558,A -85,B 0,C 180,E1 -15634.705,E2 -15634.705} C_VEL
LIN {X 0,Y 312.542,Z 444.552,A -85,B 0,C 180,E1 -15637.525,E2 -15637.525} C_VEL
LIN {X 0,Y 312.559,Z 444.677,A -85,B 0,C 180,E1 -15641.651,E2 -15641.651} C_VEL
LIN {X 0,Y 313.595,Z 448.259,A -85,B 0,C 180,E1 -15644.037,E2 -15644.037} C_VEL
LIN {X 0,Y 316.475,Z 452.236,A -85,B 0,C 180,E1 -15644.838,E2 -15644.838} C_VEL
LIN {X 0,Y 322.568,Z 461.45,A -85,B 0,C 180,E1 -15646.42,E2 -15646.42} C_VEL
LIN {X 0,Y 328.216,Z 471.244,A -85,B 0,C 180,E1 -15647.782,E2 -15647.782} C_VEL
LIN {X 0,Y 332.227,Z 479.189,A -85,B 0,C 180,E1 -15648.717,E2 -15648.717} C_VEL
LIN {X 0,Y 327.898,Z 550.851,A -85,B 0,C 180,E1 -15651.028,E2 -15651.028} C_VEL
LIN {X 0,Y 326.893,Z 565.168,A -85,B 0,C 180,E1 -15651.766,E2 -15651.766} C_VEL
LIN {X 0,Y 325.602,Z 578.165,A -85,B 0,C 180,E1 -15652.715,E2 -15652.715} C_VEL
LIN {X 0,Y 324.098,Z 589.433,A -85,B 0,C 180,E1 -15653.775,E2 -15653.775} C_VEL
LIN {X 0,Y 322.503,Z 599.768,A -85,B 0,C 180,E1 -15654.999,E2 -15654.999} C_VEL
LIN {X 0,Y 320.643,Z 610.174,A -85,B 0,C 180,E1 -15656.544,E2 -15656.544} C_VEL
LIN {X 0,Y 318.943,Z 618.738,A -85,B 0,C 180,E1 -15658.106,E2 -15658.106} C_VEL
LIN {X 0,Y 317.195,Z 627.123,A -85,B 0,C 180,E1 -15660,E2 -15660} C_VEL
LIN {X 0,Y 315.703,Z 633.798,A -85,B 0,C 180,E1 -15661.914,E2 -15661.914} C_VEL
LIN {X 0,Y 314.418,Z 639.118,A -85,B 0,C 180,E1 -15663.845,E2 -15663.845} C_VEL
LIN {X 0,Y 313.372,Z 643.23,A -85,B 0,C 180,E1 -15665.792,E2 -15665.792} C_VEL
LIN {X 0,Y 312.41,Z 646.798,A -85,B 0,C 180,E1 -15668.176,E2 -15668.176} C_VEL
LIN {X 0,Y 311.729,Z 648.708,A -85,B 0,C 180,E1 -15670.391,E2 -15670.391} C_VEL
LIN {X 0,Y 311.452,Z 649.249,A -85,B 0,C 180,E1 -15671.718,E2 -15671.718} C_VEL
LIN {X 0,Y 311.198,Z 649.21,A -85,B 0,C 180,E1 -15673.806,E2 -15673.806} C_VEL
LIN {X 0,Y 311.034,Z 648.2,A -85,B 0,C 180,E1 -15675.732,E2 -15675.732} C_VEL
LIN {X 0,Y 311.053,Z 646.948,A -85,B 0,C 180,E1 -15677.081,E2 -15677.081} C_VEL
LIN {X 0,Y 311.211,Z 644.141,A -85,B 0,C 180,E1 -15679.114,E2 -15679.114} C_VEL
LIN {X 0,Y 311.502,Z 640.135,A -85,B 0,C 180,E1 -15681.161,E2 -15681.161} C_VEL
LIN {X 0,Y 311.881,Z 634.759,A -85,B 0,C 180,E1 -15683.225,E2 -15683.225} C_VEL
LIN {X 0,Y 312.503,Z 627.861,A -85,B 0,C 180,E1 -15685.296,E2 -15685.296} C_VEL
LIN {X 0,Y 313.185,Z 620.706,A -85,B 0,C 180,E1 -15687.027,E2 -15687.027} C_VEL
LIN {X 0,Y 313.991,Z 611.91,A -85,B 0,C 180,E1 -15688.766,E2 -15688.766} C_VEL
LIN {X 0,Y 314.973,Z 600.986,A -85,B 0,C 180,E1 -15690.505,E2 -15690.505} C_VEL
LIN {X 0,Y 315.934,Z 590.11,A -85,B 0,C 180,E1 -15691.892,E2 -15691.892} C_VEL
LIN {X 0,Y 316.85,Z 577.975,A -85,B 0,C 180,E1 -15693.12,E2 -15693.12} C_VEL
LIN {X 0,Y 317.612,Z 566.014,A -85,B 0,C 180,E1 -15694.063,E2 -15694.063} C_VEL
LIN {X 0,Y 318.235,Z 552.306,A -85,B 0,C 180,E1 -15694.85,E2 -15694.85} C_VEL
LIN {X 0,Y 318.717,Z 538.421,A -85,B 0,C 180,E1 -15695.375,E2 -15695.375} C_VEL
LIN {X 0,Y 320.702,Z 467.889,A -85,B 0,C 180,E1 -15697.401,E2 -15697.401} C_VEL
LIN {X 0,Y 312.529,Z 444.56,A -85,B 0,C 180,E1 -15698.555,E2 -15698.555} C_VEL
LIN {X 0,Y 312.469,Z 444.565,A -85,B 0,C 180,E1 -15702.435,E2 -15702.435} C_VEL
LIN {X 0,Y 312.459,Z 444.563,A -85,B 0,C 180,E1 -15706.035,E2 -15706.035} C_VEL
LIN {X 0,Y 312.443,Z 444.563,A -85,B 0,C 180,E1 -15709.283,E2 -15709.283} C_VEL
LIN {X 0,Y 312.513,Z 444.557,A -85,B 0,C 180,E1 -15712.612,E2 -15712.612} C_VEL
LIN {X 0,Y 312.522,Z 444.557,A -85,B 0,C 180,E1 -15716.311,E2 -15716.311} C_VEL
LIN {X 0,Y 312.498,Z 444.561,A -85,B 0,C 180,E1 -15720.344,E2 -15720.344} C_VEL
LIN {X 0,Y 312.531,Z 444.554,A -85,B 0,C 180,E1 -15724.092,E2 -15724.092} C_VEL
LIN {X 0,Y 312.585,Z 444.545,A -85,B 0,C 180,E1 -15727.528,E2 -15727.528} C_VEL
LIN {X 0,Y 312.64,Z 444.538,A -85,B 0,C 180,E1 -15731.656,E2 -15731.656} C_VEL
LIN {X 0,Y 312.696,Z 444.531,A -85,B 0,C 180,E1 -15735.686,E2 -15735.686} C_VEL
LIN {X 0,Y 312.687,Z 444.532,A -85,B 0,C 180,E1 -15739.641,E2 -15739.641} C_VEL
LIN {X 0,Y 312.798,Z 444.522,A -85,B 0,C 180,E1 -15742.252,E2 -15742.252} C_VEL
LIN {X 0,Y 312.699,Z 444.533,A -85,B 0,C 180,E1 -15744.842,E2 -15744.842} C_VEL
LIN {X 0,Y 312.932,Z 444.501,A -85,B 0,C 180,E1 -15747.425,E2 -15747.425} C_VEL
LIN {X 0,Y 313.053,Z 444.488,A -85,B 0,C 180,E1 -15750,E2 -15750} C_VEL
